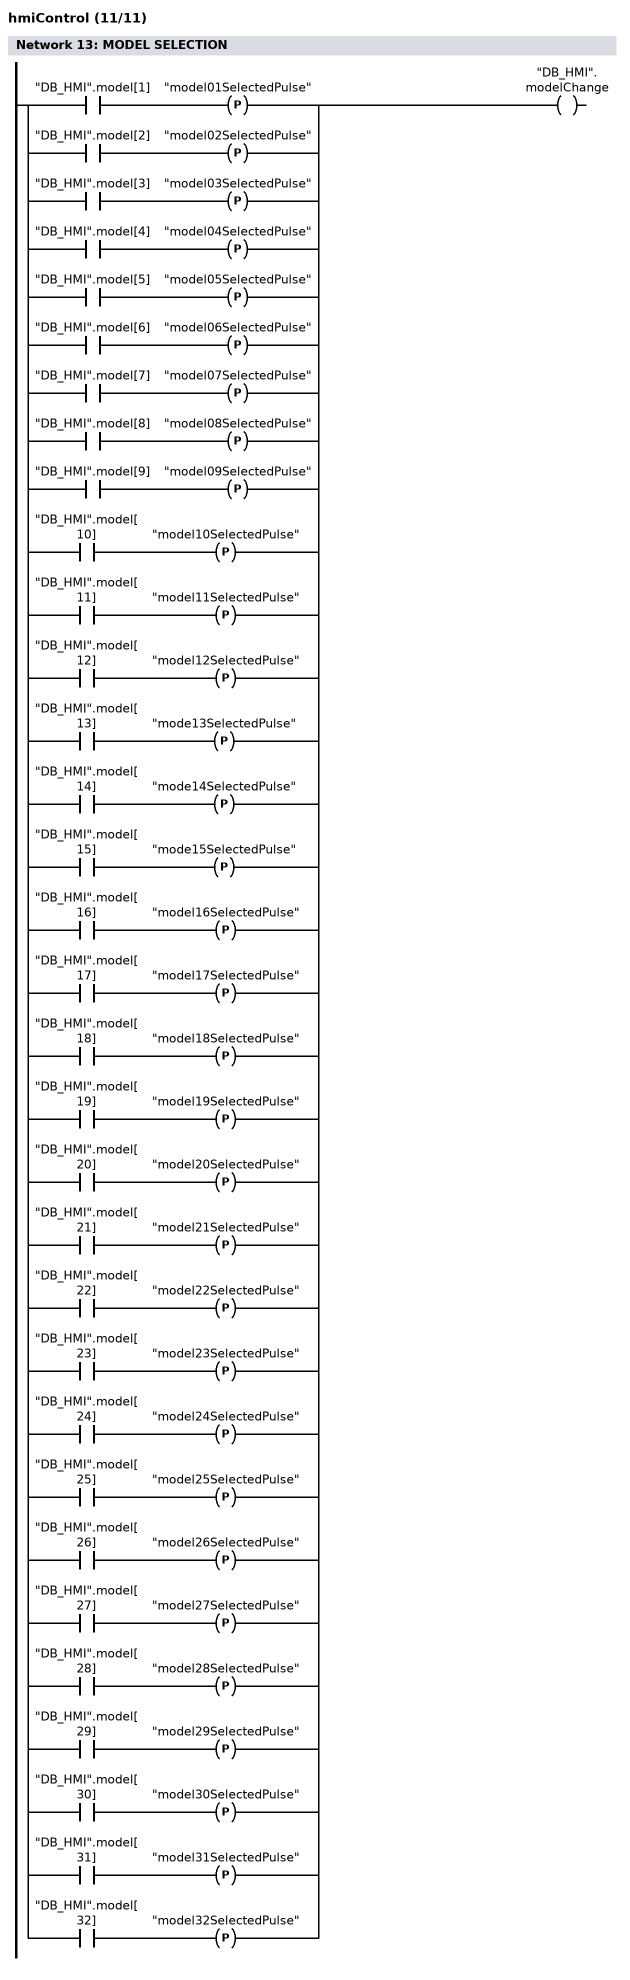
   RUNG wire#powerrail
      Contact( "DB_HMI".model[1] )
      P_Trig( "model01SelectedPulse" )
      wire#w1
      Coil( "DB_HMI".modelChange )
   END_RUNG
   RUNG wire#powerrail
      Contact( "DB_HMI".model[2] )
      P_Trig( "model02SelectedPulse" )
   END_RUNG wire#w1
   RUNG wire#powerrail
      Contact( "DB_HMI".model[3] )
      P_Trig( "model03SelectedPulse" )
   END_RUNG wire#w1
   RUNG wire#powerrail
      Contact( "DB_HMI".model[4] )
      P_Trig( "model04SelectedPulse" )
   END_RUNG wire#w1
   RUNG wire#powerrail
      Contact( "DB_HMI".model[5] )
      P_Trig( "model05SelectedPulse" )
   END_RUNG wire#w1
   RUNG wire#powerrail
      Contact( "DB_HMI".model[6] )
      P_Trig( "model06SelectedPulse" )
   END_RUNG wire#w1
   RUNG wire#powerrail
      Contact( "DB_HMI".model[7] )
      P_Trig( "model07SelectedPulse" )
   END_RUNG wire#w1
   RUNG wire#powerrail
      Contact( "DB_HMI".model[8] )
      P_Trig( "model08SelectedPulse" )
   END_RUNG wire#w1
   RUNG wire#powerrail
      Contact( "DB_HMI".model[9] )
      P_Trig( "model09SelectedPulse" )
   END_RUNG wire#w1
   RUNG wire#powerrail
      Contact( "DB_HMI".model[10] )
      P_Trig( "model10SelectedPulse" )
   END_RUNG wire#w1
   RUNG wire#powerrail
      Contact( "DB_HMI".model[11] )
      P_Trig( "model11SelectedPulse" )
   END_RUNG wire#w1
   RUNG wire#powerrail
      Contact( "DB_HMI".model[12] )
      P_Trig( "model12SelectedPulse" )
   END_RUNG wire#w1
   RUNG wire#powerrail
      Contact( "DB_HMI".model[13] )
      P_Trig( "mode13SelectedPulse" )
   END_RUNG wire#w1
   RUNG wire#powerrail
      Contact( "DB_HMI".model[14] )
      P_Trig( "mode14SelectedPulse" )
   END_RUNG wire#w1
   RUNG wire#powerrail
      Contact( "DB_HMI".model[15] )
      P_Trig( "mode15SelectedPulse" )
   END_RUNG wire#w1
   RUNG wire#powerrail
      Contact( "DB_HMI".model[16] )
      P_Trig( "model16SelectedPulse" )
   END_RUNG wire#w1
   RUNG wire#powerrail
      Contact( "DB_HMI".model[17] )
      P_Trig( "model17SelectedPulse" )
   END_RUNG wire#w1
   RUNG wire#powerrail
      Contact( "DB_HMI".model[18] )
      P_Trig( "model18SelectedPulse" )
   END_RUNG wire#w1
   RUNG wire#powerrail
      Contact( "DB_HMI".model[19] )
      P_Trig( "model19SelectedPulse" )
   END_RUNG wire#w1
   RUNG wire#powerrail
      Contact( "DB_HMI".model[20] )
      P_Trig( "model20SelectedPulse" )
   END_RUNG wire#w1
   RUNG wire#powerrail
      Contact( "DB_HMI".model[21] )
      P_Trig( "model21SelectedPulse" )
   END_RUNG wire#w1
   RUNG wire#powerrail
      Contact( "DB_HMI".model[22] )
      P_Trig( "model22SelectedPulse" )
   END_RUNG wire#w1
   RUNG wire#powerrail
      Contact( "DB_HMI".model[23] )
      P_Trig( "model23SelectedPulse" )
   END_RUNG wire#w1
   RUNG wire#powerrail
      Contact( "DB_HMI".model[24] )
      P_Trig( "model24SelectedPulse" )
   END_RUNG wire#w1
   RUNG wire#powerrail
      Contact( "DB_HMI".model[25] )
      P_Trig( "model25SelectedPulse" )
   END_RUNG wire#w1
   RUNG wire#powerrail
      Contact( "DB_HMI".model[26] )
      P_Trig( "model26SelectedPulse" )
   END_RUNG wire#w1
   RUNG wire#powerrail
      Contact( "DB_HMI".model[27] )
      P_Trig( "model27SelectedPulse" )
   END_RUNG wire#w1
   RUNG wire#powerrail
      Contact( "DB_HMI".model[28] )
      P_Trig( "model28SelectedPulse" )
   END_RUNG wire#w1
   RUNG wire#powerrail
      Contact( "DB_HMI".model[29] )
      P_Trig( "model29SelectedPulse" )
   END_RUNG wire#w1
   RUNG wire#powerrail
      Contact( "DB_HMI".model[30] )
      P_Trig( "model30SelectedPulse" )
   END_RUNG wire#w1
   RUNG wire#powerrail
      Contact( "DB_HMI".model[31] )
      P_Trig( "model31SelectedPulse" )
   END_RUNG wire#w1
   RUNG wire#powerrail
      Contact( "DB_HMI".model[32] )
      P_Trig( "model32SelectedPulse" )
   END_RUNG wire#w1
   // the same network as SCL:
   #_w1 := "DB_HMI".model[1] AND NOT "model01SelectedPulse";   // rising edge
   "model01SelectedPulse" := "DB_HMI".model[1];
   #_w2 := "DB_HMI".model[2] AND NOT "model02SelectedPulse";   // rising edge
   "model02SelectedPulse" := "DB_HMI".model[2];
   #_w3 := "DB_HMI".model[3] AND NOT "model03SelectedPulse";   // rising edge
   "model03SelectedPulse" := "DB_HMI".model[3];
   #_w4 := "DB_HMI".model[4] AND NOT "model04SelectedPulse";   // rising edge
   "model04SelectedPulse" := "DB_HMI".model[4];
   #_w5 := "DB_HMI".model[5] AND NOT "model05SelectedPulse";   // rising edge
   "model05SelectedPulse" := "DB_HMI".model[5];
   #_w6 := "DB_HMI".model[6] AND NOT "model06SelectedPulse";   // rising edge
   "model06SelectedPulse" := "DB_HMI".model[6];
   #_w7 := "DB_HMI".model[7] AND NOT "model07SelectedPulse";   // rising edge
   "model07SelectedPulse" := "DB_HMI".model[7];
   #_w8 := "DB_HMI".model[8] AND NOT "model08SelectedPulse";   // rising edge
   "model08SelectedPulse" := "DB_HMI".model[8];
   #_w9 := "DB_HMI".model[9] AND NOT "model09SelectedPulse";   // rising edge
   "model09SelectedPulse" := "DB_HMI".model[9];
   #_w10 := "DB_HMI".model[10] AND NOT "model10SelectedPulse";   // rising edge
   "model10SelectedPulse" := "DB_HMI".model[10];
   #_w11 := "DB_HMI".model[11] AND NOT "model11SelectedPulse";   // rising edge
   "model11SelectedPulse" := "DB_HMI".model[11];
   #_w12 := "DB_HMI".model[12] AND NOT "model12SelectedPulse";   // rising edge
   "model12SelectedPulse" := "DB_HMI".model[12];
   #_w13 := "DB_HMI".model[13] AND NOT "mode13SelectedPulse";   // rising edge
   "mode13SelectedPulse" := "DB_HMI".model[13];
   #_w14 := "DB_HMI".model[14] AND NOT "mode14SelectedPulse";   // rising edge
   "mode14SelectedPulse" := "DB_HMI".model[14];
   #_w15 := "DB_HMI".model[15] AND NOT "mode15SelectedPulse";   // rising edge
   "mode15SelectedPulse" := "DB_HMI".model[15];
   #_w16 := "DB_HMI".model[16] AND NOT "model16SelectedPulse";   // rising edge
   "model16SelectedPulse" := "DB_HMI".model[16];
   #_w17 := "DB_HMI".model[17] AND NOT "model17SelectedPulse";   // rising edge
   "model17SelectedPulse" := "DB_HMI".model[17];
   #_w18 := "DB_HMI".model[18] AND NOT "model18SelectedPulse";   // rising edge
   "model18SelectedPulse" := "DB_HMI".model[18];
   #_w19 := "DB_HMI".model[19] AND NOT "model19SelectedPulse";   // rising edge
   "model19SelectedPulse" := "DB_HMI".model[19];
   #_w20 := "DB_HMI".model[20] AND NOT "model20SelectedPulse";   // rising edge
   "model20SelectedPulse" := "DB_HMI".model[20];
   #_w21 := "DB_HMI".model[21] AND NOT "model21SelectedPulse";   // rising edge
   "model21SelectedPulse" := "DB_HMI".model[21];
   #_w22 := "DB_HMI".model[22] AND NOT "model22SelectedPulse";   // rising edge
   "model22SelectedPulse" := "DB_HMI".model[22];
   #_w23 := "DB_HMI".model[23] AND NOT "model23SelectedPulse";   // rising edge
   "model23SelectedPulse" := "DB_HMI".model[23];
   #_w24 := "DB_HMI".model[24] AND NOT "model24SelectedPulse";   // rising edge
   "model24SelectedPulse" := "DB_HMI".model[24];
   #_w25 := "DB_HMI".model[25] AND NOT "model25SelectedPulse";   // rising edge
   "model25SelectedPulse" := "DB_HMI".model[25];
   #_w26 := "DB_HMI".model[26] AND NOT "model26SelectedPulse";   // rising edge
   "model26SelectedPulse" := "DB_HMI".model[26];
   #_w27 := "DB_HMI".model[27] AND NOT "model27SelectedPulse";   // rising edge
   "model27SelectedPulse" := "DB_HMI".model[27];
   #_w28 := "DB_HMI".model[28] AND NOT "model28SelectedPulse";   // rising edge
   "model28SelectedPulse" := "DB_HMI".model[28];
   #_w29 := "DB_HMI".model[29] AND NOT "model29SelectedPulse";   // rising edge
   "model29SelectedPulse" := "DB_HMI".model[29];
   #_w30 := "DB_HMI".model[30] AND NOT "model30SelectedPulse";   // rising edge
   "model30SelectedPulse" := "DB_HMI".model[30];
   #_w31 := "DB_HMI".model[31] AND NOT "model31SelectedPulse";   // rising edge
   "model31SelectedPulse" := "DB_HMI".model[31];
   #_w32 := "DB_HMI".model[32] AND NOT "model32SelectedPulse";   // rising edge
   "model32SelectedPulse" := "DB_HMI".model[32];
   "DB_HMI".modelChange := #_w1 OR #_w2 OR #_w3 OR #_w4 OR #_w5 OR #_w6 OR #_w7 OR #_w8 OR #_w9 OR #_w10 OR #_w11 OR #_w12 OR #_w13 OR #_w14 OR #_w15 OR #_w16 OR #_w17 OR #_w18 OR #_w19 OR #_w20 OR #_w21 OR #_w22 OR #_w23 OR #_w24 OR #_w25 OR #_w26 OR #_w27 OR #_w28 OR #_w29 OR #_w30 OR #_w31 OR #_w32;
END_REGION
END_FUNCTION

FUNCTION "MODE" : Void   // FC4, LAD
{ S7_Optimized_Access := 'TRUE' }
VERSION : 0.1
// stored: AutoNumber true, IsIECCheckEnabled false, SetENOAutomatically false, UDAEnableTagReadback false
   VAR_TEMP
      f7 : Bool;
      BF7 : Bool;
   END_VAR
BEGIN

REGION Network 1: MODE CHANGE
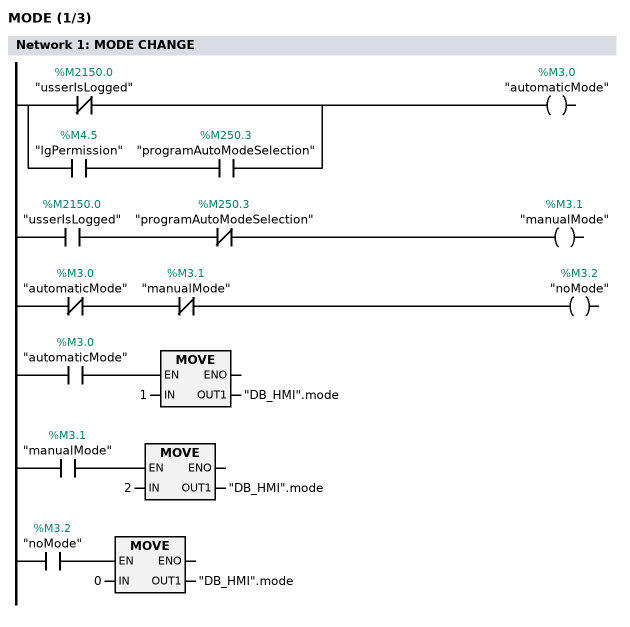
   RUNG wire#powerrail
      I_Contact( "usserIsLogged" )
      wire#w1
      Coil( "automaticMode" )
   END_RUNG
   RUNG wire#powerrail
      Contact( "lgPermission" )
      Contact( "programAutoModeSelection" )
   END_RUNG wire#w1
   RUNG wire#powerrail
      Contact( "usserIsLogged" )
      I_Contact( "programAutoModeSelection" )
      Coil( "manualMode" )
   END_RUNG
   RUNG wire#powerrail
      I_Contact( "automaticMode" )
      I_Contact( "manualMode" )
      Coil( "noMode" )
   END_RUNG
   RUNG wire#powerrail
      Contact( "automaticMode" )
      Move(in := 1, out1 => "DB_HMI".mode)
   END_RUNG
   RUNG wire#powerrail
      Contact( "manualMode" )
      Move(in := 2, out1 => "DB_HMI".mode)
   END_RUNG
   RUNG wire#powerrail
      Contact( "noMode" )
      Move(in := 0, out1 => "DB_HMI".mode)
   END_RUNG
   // the same network as SCL:
   "automaticMode" := NOT "usserIsLogged" OR ("lgPermission" AND "programAutoModeSelection");
   "manualMode" := "usserIsLogged" AND NOT "programAutoModeSelection";
   "noMode" := NOT "automaticMode" AND NOT "manualMode";
   IF "automaticMode" THEN "DB_HMI".mode := 1; END_IF;
   IF "manualMode" THEN "DB_HMI".mode := 2; END_IF;
   IF "noMode" THEN "DB_HMI".mode := 0; END_IF;
END_REGION

REGION Network 2: MODEL SELECTION
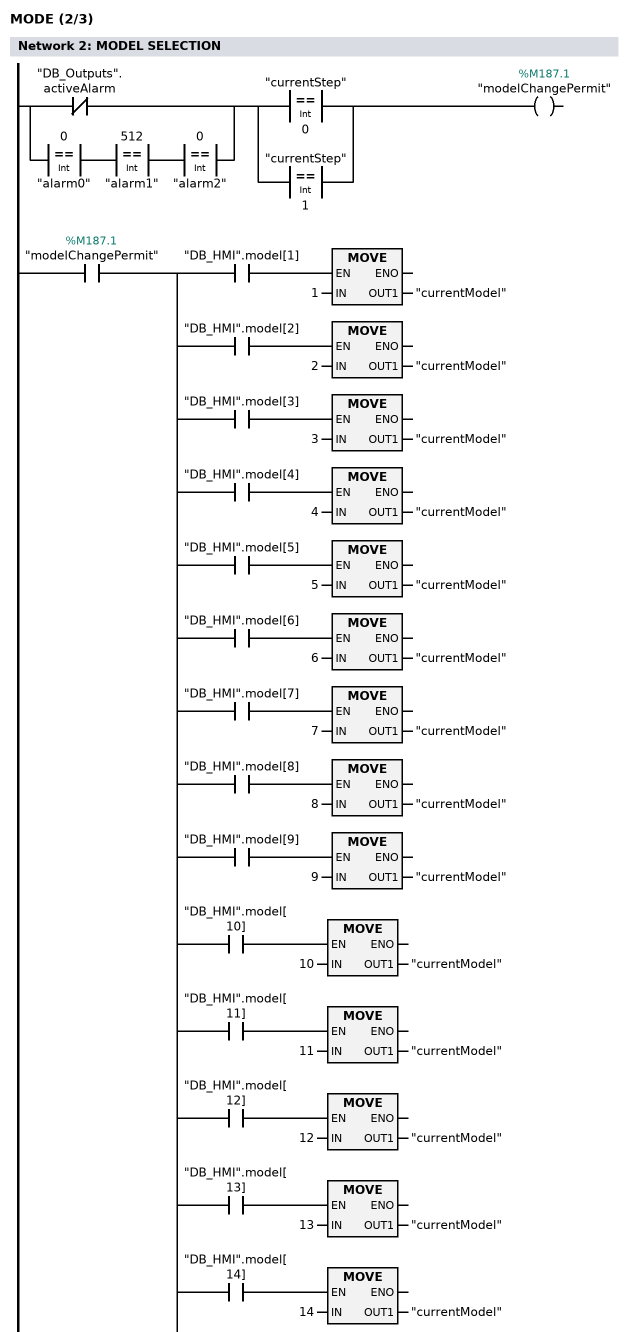
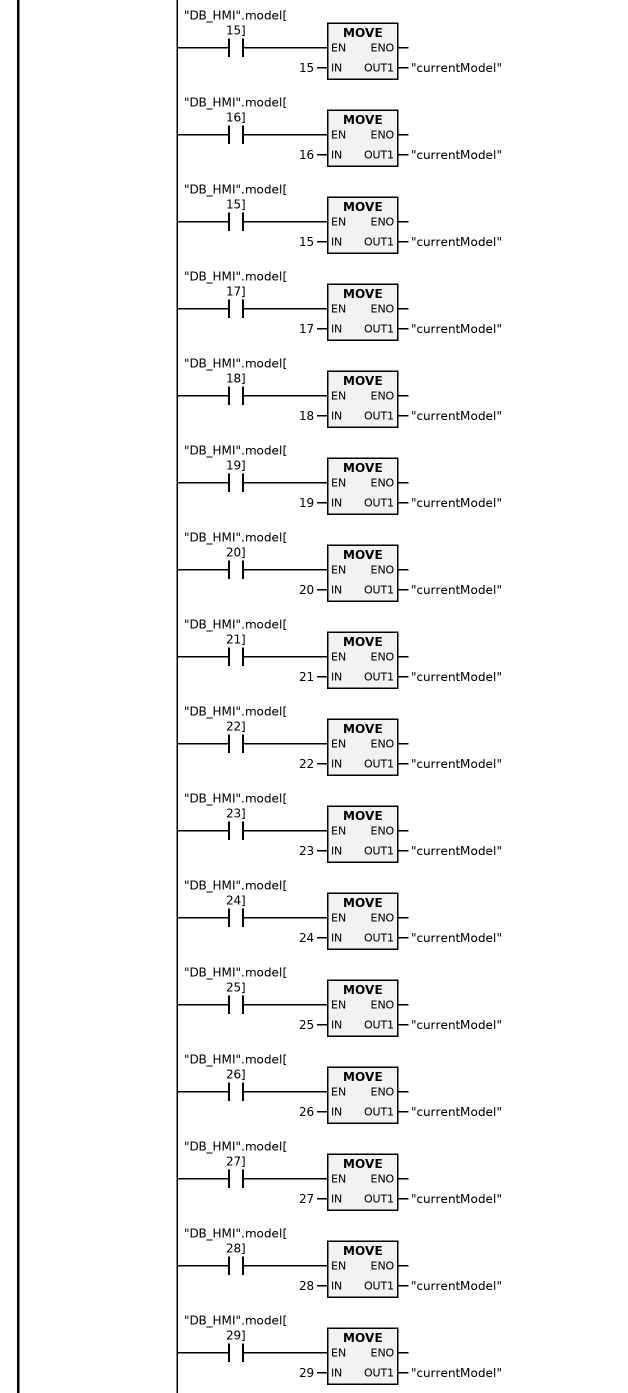
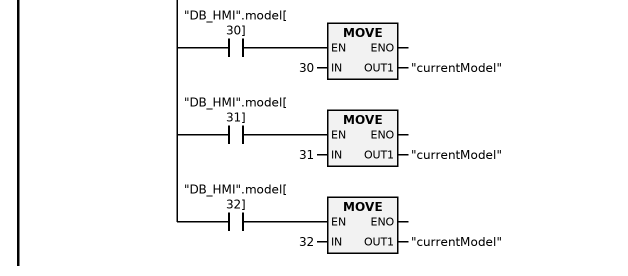
   RUNG wire#powerrail
      I_Contact( "DB_Outputs".activeAlarm )
      wire#w1
      { S7_Templates := "SrcType := Int" } EQ_Contact(in1 := "currentStep", in2 := 0)
      wire#w2
      Coil( "modelChangePermit" )
   END_RUNG
   RUNG wire#powerrail
      { S7_Templates := "SrcType := Int" } EQ_Contact(in1 := 0, in2 := "alarm0")
      { S7_Templates := "SrcType := Int" } EQ_Contact(in1 := 512, in2 := "alarm1")
      { S7_Templates := "SrcType := Int" } EQ_Contact(in1 := 0, in2 := "alarm2")
   END_RUNG wire#w1
   RUNG wire#w1
      { S7_Templates := "SrcType := Int" } EQ_Contact(in1 := "currentStep", in2 := 1)
   END_RUNG wire#w2
   RUNG wire#powerrail
      Contact( "modelChangePermit" )
      wire#w3
      Contact( "DB_HMI".model[1] )
      Move(in := 1, out1 => "currentModel")
   END_RUNG
   RUNG wire#w3
      Contact( "DB_HMI".model[2] )
      Move(in := 2, out1 => "currentModel")
   END_RUNG
   RUNG wire#w3
      Contact( "DB_HMI".model[3] )
      Move(in := 3, out1 => "currentModel")
   END_RUNG
   RUNG wire#w3
      Contact( "DB_HMI".model[4] )
      Move(in := 4, out1 => "currentModel")
   END_RUNG
   RUNG wire#w3
      Contact( "DB_HMI".model[5] )
      Move(in := 5, out1 => "currentModel")
   END_RUNG
   RUNG wire#w3
      Contact( "DB_HMI".model[6] )
      Move(in := 6, out1 => "currentModel")
   END_RUNG
   RUNG wire#w3
      Contact( "DB_HMI".model[7] )
      Move(in := 7, out1 => "currentModel")
   END_RUNG
   RUNG wire#w3
      Contact( "DB_HMI".model[8] )
      Move(in := 8, out1 => "currentModel")
   END_RUNG
   RUNG wire#w3
      Contact( "DB_HMI".model[9] )
      Move(in := 9, out1 => "currentModel")
   END_RUNG
   RUNG wire#w3
      Contact( "DB_HMI".model[10] )
      Move(in := 10, out1 => "currentModel")
   END_RUNG
   RUNG wire#w3
      Contact( "DB_HMI".model[11] )
      Move(in := 11, out1 => "currentModel")
   END_RUNG
   RUNG wire#w3
      Contact( "DB_HMI".model[12] )
      Move(in := 12, out1 => "currentModel")
   END_RUNG
   RUNG wire#w3
      Contact( "DB_HMI".model[13] )
      Move(in := 13, out1 => "currentModel")
   END_RUNG
   RUNG wire#w3
      Contact( "DB_HMI".model[14] )
      Move(in := 14, out1 => "currentModel")
   END_RUNG
   RUNG wire#w3
      Contact( "DB_HMI".model[15] )
      Move(in := 15, out1 => "currentModel")
   END_RUNG
   RUNG wire#w3
      Contact( "DB_HMI".model[16] )
      Move(in := 16, out1 => "currentModel")
   END_RUNG
   RUNG wire#w3
      Contact( "DB_HMI".model[15] )
      Move(in := 15, out1 => "currentModel")
   END_RUNG
   RUNG wire#w3
      Contact( "DB_HMI".model[17] )
      Move(in := 17, out1 => "currentModel")
   END_RUNG
   RUNG wire#w3
      Contact( "DB_HMI".model[18] )
      Move(in := 18, out1 => "currentModel")
   END_RUNG
   RUNG wire#w3
      Contact( "DB_HMI".model[19] )
      Move(in := 19, out1 => "currentModel")
   END_RUNG
   RUNG wire#w3
      Contact( "DB_HMI".model[20] )
      Move(in := 20, out1 => "currentModel")
   END_RUNG
   RUNG wire#w3
      Contact( "DB_HMI".model[21] )
      Move(in := 21, out1 => "currentModel")
   END_RUNG
   RUNG wire#w3
      Contact( "DB_HMI".model[22] )
      Move(in := 22, out1 => "currentModel")
   END_RUNG
   RUNG wire#w3
      Contact( "DB_HMI".model[23] )
      Move(in := 23, out1 => "currentModel")
   END_RUNG
   RUNG wire#w3
      Contact( "DB_HMI".model[24] )
      Move(in := 24, out1 => "currentModel")
   END_RUNG
   RUNG wire#w3
      Contact( "DB_HMI".model[25] )
      Move(in := 25, out1 => "currentModel")
   END_RUNG
   RUNG wire#w3
      Contact( "DB_HMI".model[26] )
      Move(in := 26, out1 => "currentModel")
   END_RUNG
   RUNG wire#w3
      Contact( "DB_HMI".model[27] )
      Move(in := 27, out1 => "currentModel")
   END_RUNG
   RUNG wire#w3
      Contact( "DB_HMI".model[28] )
      Move(in := 28, out1 => "currentModel")
   END_RUNG
   RUNG wire#w3
      Contact( "DB_HMI".model[29] )
      Move(in := 29, out1 => "currentModel")
   END_RUNG
   RUNG wire#w3
      Contact( "DB_HMI".model[30] )
      Move(in := 30, out1 => "currentModel")
   END_RUNG
   RUNG wire#w3
      Contact( "DB_HMI".model[31] )
      Move(in := 31, out1 => "currentModel")
   END_RUNG
   RUNG wire#w3
      Contact( "DB_HMI".model[32] )
      Move(in := 32, out1 => "currentModel")
   END_RUNG
   // the same network as SCL:
   "modelChangePermit" := (NOT "DB_Outputs".activeAlarm OR ((0 = "alarm0") AND (512 = "alarm1") AND (0 = "alarm2"))) AND (("currentStep" = 0) OR ("currentStep" = 1));
   IF "modelChangePermit" AND "DB_HMI".model[1] THEN "currentModel" := 1; END_IF;
   IF "modelChangePermit" AND "DB_HMI".model[2] THEN "currentModel" := 2; END_IF;
   IF "modelChangePermit" AND "DB_HMI".model[3] THEN "currentModel" := 3; END_IF;
   IF "modelChangePermit" AND "DB_HMI".model[4] THEN "currentModel" := 4; END_IF;
   IF "modelChangePermit" AND "DB_HMI".model[5] THEN "currentModel" := 5; END_IF;
   IF "modelChangePermit" AND "DB_HMI".model[6] THEN "currentModel" := 6; END_IF;
   IF "modelChangePermit" AND "DB_HMI".model[7] THEN "currentModel" := 7; END_IF;
   IF "modelChangePermit" AND "DB_HMI".model[8] THEN "currentModel" := 8; END_IF;
   IF "modelChangePermit" AND "DB_HMI".model[9] THEN "currentModel" := 9; END_IF;
   IF "modelChangePermit" AND "DB_HMI".model[10] THEN "currentModel" := 10; END_IF;
   IF "modelChangePermit" AND "DB_HMI".model[11] THEN "currentModel" := 11; END_IF;
   IF "modelChangePermit" AND "DB_HMI".model[12] THEN "currentModel" := 12; END_IF;
   IF "modelChangePermit" AND "DB_HMI".model[13] THEN "currentModel" := 13; END_IF;
   IF "modelChangePermit" AND "DB_HMI".model[14] THEN "currentModel" := 14; END_IF;
   IF "modelChangePermit" AND "DB_HMI".model[15] THEN "currentModel" := 15; END_IF;
   IF "modelChangePermit" AND "DB_HMI".model[16] THEN "currentModel" := 16; END_IF;
   IF "modelChangePermit" AND "DB_HMI".model[15] THEN "currentModel" := 15; END_IF;
   IF "modelChangePermit" AND "DB_HMI".model[17] THEN "currentModel" := 17; END_IF;
   IF "modelChangePermit" AND "DB_HMI".model[18] THEN "currentModel" := 18; END_IF;
   IF "modelChangePermit" AND "DB_HMI".model[19] THEN "currentModel" := 19; END_IF;
   IF "modelChangePermit" AND "DB_HMI".model[20] THEN "currentModel" := 20; END_IF;
   IF "modelChangePermit" AND "DB_HMI".model[21] THEN "currentModel" := 21; END_IF;
   IF "modelChangePermit" AND "DB_HMI".model[22] THEN "currentModel" := 22; END_IF;
   IF "modelChangePermit" AND "DB_HMI".model[23] THEN "currentModel" := 23; END_IF;
   IF "modelChangePermit" AND "DB_HMI".model[24] THEN "currentModel" := 24; END_IF;
   IF "modelChangePermit" AND "DB_HMI".model[25] THEN "currentModel" := 25; END_IF;
   IF "modelChangePermit" AND "DB_HMI".model[26] THEN "currentModel" := 26; END_IF;
   IF "modelChangePermit" AND "DB_HMI".model[27] THEN "currentModel" := 27; END_IF;
   IF "modelChangePermit" AND "DB_HMI".model[28] THEN "currentModel" := 28; END_IF;
   IF "modelChangePermit" AND "DB_HMI".model[29] THEN "currentModel" := 29; END_IF;
   IF "modelChangePermit" AND "DB_HMI".model[30] THEN "currentModel" := 30; END_IF;
   IF "modelChangePermit" AND "DB_HMI".model[31] THEN "currentModel" := 31; END_IF;
   IF "modelChangePermit" AND "DB_HMI".model[32] THEN "currentModel" := 32; END_IF;
END_REGION

REGION Network 3: GAP LEADER HMI MODE
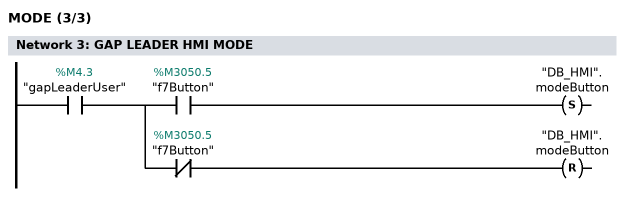
   RUNG wire#powerrail
      Contact( "gapLeaderUser" )
      wire#w1
      Contact( "f7Button" )
      S_Coil( "DB_HMI".modeButton )
   END_RUNG
   RUNG wire#w1
      I_Contact( "f7Button" )
      R_Coil( "DB_HMI".modeButton )
   END_RUNG
   // the same network as SCL:
   IF "gapLeaderUser" AND "f7Button" THEN "DB_HMI".modeButton := TRUE; END_IF;
   IF "gapLeaderUser" AND NOT "f7Button" THEN "DB_HMI".modeButton := FALSE; END_IF;
END_REGION
END_FUNCTION

FUNCTION "MISC" : Void   // FC5, LAD
{ S7_Optimized_Access := 'TRUE' }
VERSION : 0.1
// stored: AutoNumber true, IsIECCheckEnabled false, SetENOAutomatically false, UDAEnableTagReadback false
   VAR_TEMP
      INTERMITENTE : Bool;
      RESETEADO : Bool;
      RESULT_2 : UInt;
      Result_3 : Int;
   END_VAR
   VAR_TEMP   // added for the SCL form of the ladder/FBD networks
      _w1 : Bool;
      _w2 : Bool;
      _w3 : Bool;
      _w4 : Bool;
   END_VAR
BEGIN

REGION Network 1: HMI OPTIONS BUTTON SHUTOFF
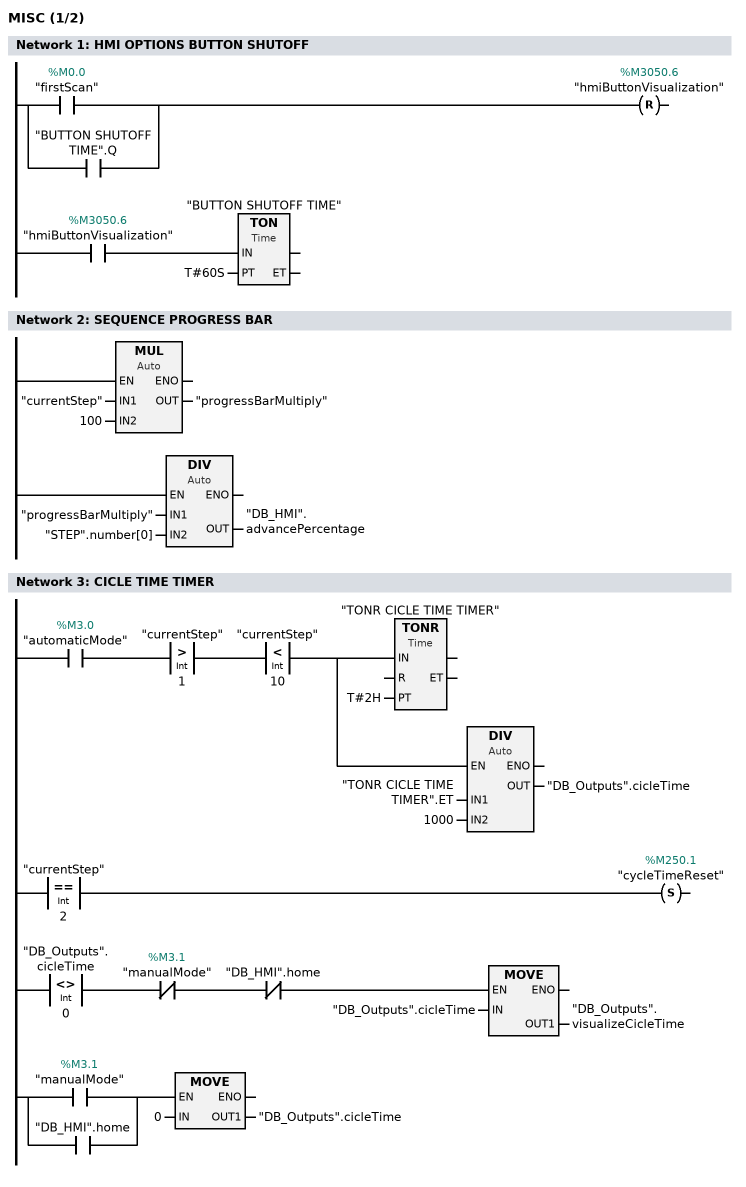
   RUNG wire#powerrail
      Contact( "firstScan" )
      wire#w1
      R_Coil( "hmiButtonVisualization" )
   END_RUNG
   RUNG wire#powerrail
      Contact( "BUTTON SHUTOFF TIME".Q )
   END_RUNG wire#w1
   RUNG wire#powerrail
      Contact( "hmiButtonVisualization" )
      { S7_Templates := "time_type := Time" } "BUTTON SHUTOFF TIME".TON(pt := T#60S, et =>)
   END_RUNG
   // the same network as SCL:
   IF "firstScan" OR "BUTTON SHUTOFF TIME".Q THEN "hmiButtonVisualization" := FALSE; END_IF;
   "BUTTON SHUTOFF TIME".TON(IN := "hmiButtonVisualization", PT := T#60S);
END_REGION

REGION Network 2: SEQUENCE PROGRESS BAR
   RUNG wire#powerrail
      Mul(in1 := "currentStep", in2 := 100, out => "progressBarMultiply")
   END_RUNG
   RUNG wire#powerrail
      Div(in1 := "progressBarMultiply", in2 := "STEP".number[0], out => "DB_HMI".advancePercentage)
   END_RUNG
   // the same network as SCL:
   "progressBarMultiply" := "currentStep" * 100;
   "DB_HMI".advancePercentage := "progressBarMultiply" / "STEP".number[0];
END_REGION

REGION Network 3: CICLE TIME TIMER
   RUNG wire#powerrail
      Contact( "automaticMode" )
      { S7_Templates := "SrcType := Int" } GT_Contact(in1 := "currentStep", in2 := 1)
      { S7_Templates := "SrcType := Int" } LT_Contact(in1 := "currentStep", in2 := 10)
      wire#w1
      { S7_Templates := "time_type := Time" } "TONR CICLE TIME TIMER".TONR(r :=, pt := T#2H, et =>)
   END_RUNG
   RUNG wire#w1
      Div(in1 := "TONR CICLE TIME TIMER".ET, in2 := 1000, out => "DB_Outputs".cicleTime)
   END_RUNG
   RUNG wire#powerrail
      { S7_Templates := "SrcType := Int" } EQ_Contact(in1 := "currentStep", in2 := 2)
      S_Coil( "cycleTimeReset" )
   END_RUNG
   RUNG wire#powerrail
      { S7_Templates := "SrcType := Int" } NE_Contact(in1 := "DB_Outputs".cicleTime, in2 := 0)
      I_Contact( "manualMode" )
      I_Contact( "DB_HMI".home )
      Move(in := "DB_Outputs".cicleTime, out1 => "DB_Outputs".visualizeCicleTime)
   END_RUNG
   RUNG wire#powerrail
      Contact( "manualMode" )
      wire#w2
      Move(in := 0, out1 => "DB_Outputs".cicleTime)
   END_RUNG
   RUNG wire#powerrail
      Contact( "DB_HMI".home )
   END_RUNG wire#w2
   // the same network as SCL:
   #_w1 := "automaticMode" AND ("currentStep" > 1) AND ("currentStep" < 10);
   "TONR CICLE TIME TIMER".TONR(IN := #_w1, PT := T#2H);
   IF #_w1 THEN "DB_Outputs".cicleTime := "TONR CICLE TIME TIMER".ET / 1000; END_IF;
   IF "currentStep" = 2 THEN "cycleTimeReset" := TRUE; END_IF;
   IF ("DB_Outputs".cicleTime <> 0) AND NOT "manualMode" AND NOT "DB_HMI".home THEN
       "DB_Outputs".visualizeCicleTime := "DB_Outputs".cicleTime;
   END_IF;
   IF "manualMode" OR "DB_HMI".home THEN "DB_Outputs".cicleTime := 0; END_IF;
END_REGION

REGION Network 4: STEP CHANGE TIMER
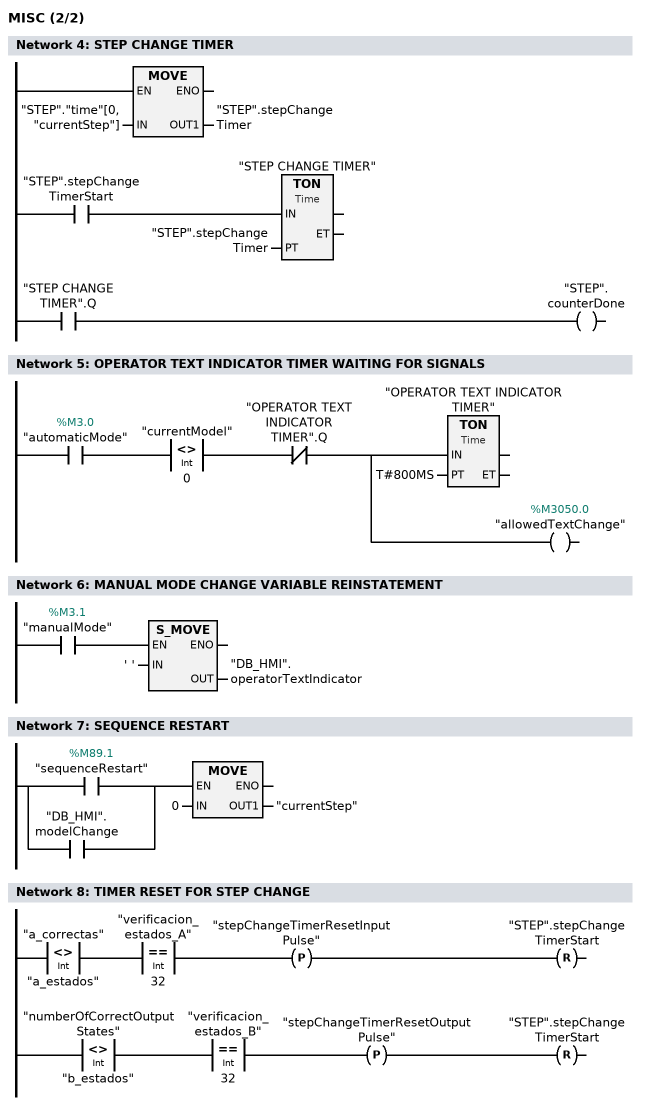
   RUNG wire#powerrail
      Move(in := "STEP"."time"[0, "currentStep"], out1 => "STEP".stepChangeTimer)
   END_RUNG
   RUNG wire#powerrail
      Contact( "STEP".stepChangeTimerStart )
      { S7_Templates := "time_type := Time" } "STEP CHANGE TIMER".TON(pt := "STEP".stepChangeTimer, et =>)
   END_RUNG
   RUNG wire#powerrail
      Contact( "STEP CHANGE TIMER".Q )
      Coil( "STEP".counterDone )
   END_RUNG
   // the same network as SCL:
   "STEP".stepChangeTimer := "STEP"."time"[0, "currentStep"];
   "STEP CHANGE TIMER".TON(IN := "STEP".stepChangeTimerStart, PT := "STEP".stepChangeTimer);
   "STEP".counterDone := "STEP CHANGE TIMER".Q;
END_REGION

REGION Network 5: OPERATOR TEXT INDICATOR TIMER WAITING FOR SIGNALS
   RUNG wire#powerrail
      Contact( "automaticMode" )
      { S7_Templates := "SrcType := Int" } NE_Contact(in1 := "currentModel", in2 := 0)
      I_Contact( "OPERATOR TEXT INDICATOR TIMER".Q )
      wire#w1
      { S7_Templates := "time_type := Time" } "OPERATOR TEXT INDICATOR TIMER".TON(pt := T#800MS, et =>)
   END_RUNG
   RUNG wire#w1
      Coil( "allowedTextChange" )
   END_RUNG
   // the same network as SCL:
   #_w1 := "automaticMode" AND ("currentModel" <> 0) AND NOT "OPERATOR TEXT INDICATOR TIMER".Q;
   "OPERATOR TEXT INDICATOR TIMER".TON(IN := #_w1, PT := T#800MS);
   "allowedTextChange" := #_w1;
END_REGION

REGION Network 6: MANUAL MODE CHANGE VARIABLE REINSTATEMENT
   RUNG wire#powerrail
      Contact( "manualMode" )
      S_Move(in := ' ', out => "DB_HMI".operatorTextIndicator)
   END_RUNG
   // the same network as SCL:
   IF "manualMode" THEN "DB_HMI".operatorTextIndicator := ' '; END_IF;
END_REGION

REGION Network 7: SEQUENCE RESTART
   RUNG wire#powerrail
      Contact( "sequenceRestart" )
      wire#w1
      Move(in := 0, out1 => "currentStep")
   END_RUNG
   RUNG wire#powerrail
      Contact( "DB_HMI".modelChange )
   END_RUNG wire#w1
   // the same network as SCL:
   IF "sequenceRestart" OR "DB_HMI".modelChange THEN "currentStep" := 0; END_IF;
END_REGION

REGION Network 8: TIMER RESET FOR STEP CHANGE
   RUNG wire#powerrail
      { S7_Templates := "SrcType := Int" } NE_Contact(in1 := "a_correctas", in2 := "a_estados")
      { S7_Templates := "SrcType := Int" } EQ_Contact(in1 := "verificacion_estados_A", in2 := 32)
      P_Trig( "stepChangeTimerResetInputPulse" )
      R_Coil( "STEP".stepChangeTimerStart )
   END_RUNG
   RUNG wire#powerrail
      { S7_Templates := "SrcType := Int" } NE_Contact(in1 := "numberOfCorrectOutputStates", in2 := "b_estados")
      { S7_Templates := "SrcType := Int" } EQ_Contact(in1 := "verificacion_estados_B", in2 := 32)
      P_Trig( "stepChangeTimerResetOutputPulse" )
      R_Coil( "STEP".stepChangeTimerStart )
   END_RUNG
   // the same network as SCL:
   #_w1 := ("a_correctas" <> "a_estados") AND ("verificacion_estados_A" = 32);
   #_w2 := #_w1 AND NOT "stepChangeTimerResetInputPulse";   // rising edge
   "stepChangeTimerResetInputPulse" := #_w1;
   IF #_w2 THEN "STEP".stepChangeTimerStart := FALSE; END_IF;
   #_w3 := ("numberOfCorrectOutputStates" <> "b_estados") AND ("verificacion_estados_B" = 32);
   #_w4 := #_w3 AND NOT "stepChangeTimerResetOutputPulse";   // rising edge
   "stepChangeTimerResetOutputPulse" := #_w3;
   IF #_w4 THEN "STEP".stepChangeTimerStart := FALSE; END_IF;
END_REGION
END_FUNCTION

FUNCTION "MODIFY RECIPE" : Void   // FC6, LAD
{ S7_Optimized_Access := 'TRUE' }
VERSION : 0.1
// stored: AutoNumber true, IsIECCheckEnabled false, SetENOAutomatically false, UDAEnableTagReadback false
   VAR_TEMP   // added for the SCL form of the ladder/FBD networks
      _w1 : Bool;
      _w2 : Bool;
   END_VAR
BEGIN

REGION Network 1: ERASE A STEP
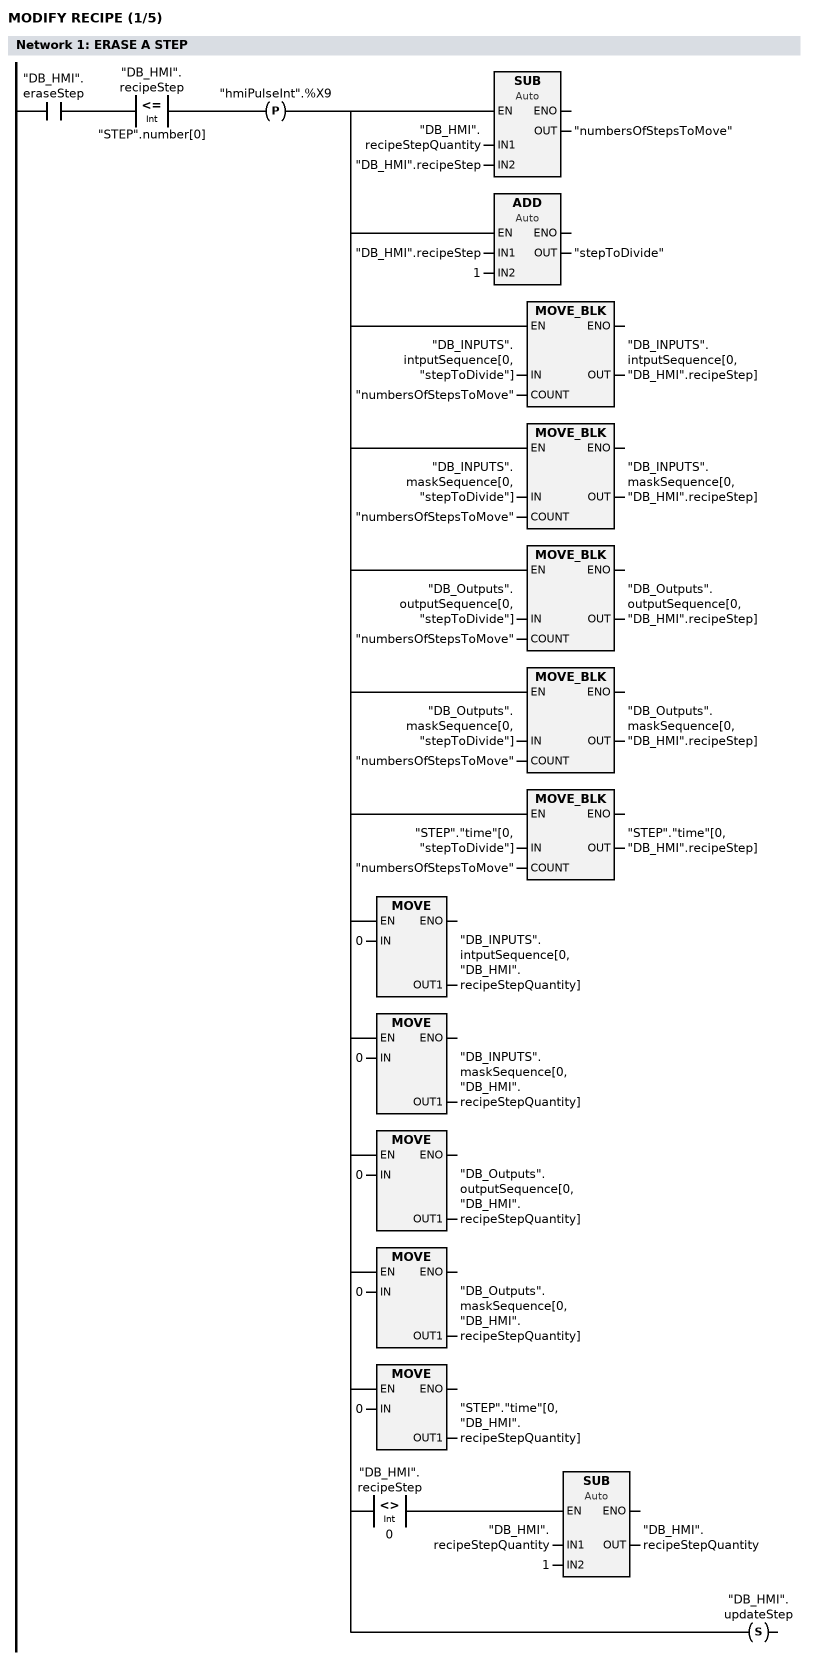
   #_w1 := "DB_HMI".eraseStep AND ("DB_HMI".recipeStep <= "STEP".number[0]);
   #_w2 := #_w1 AND NOT "hmiPulseInt".%X9;   // rising edge
   "hmiPulseInt".%X9 := #_w1;
   IF #_w2 THEN
       "numbersOfStepsToMove" := "DB_HMI".recipeStepQuantity - "DB_HMI".recipeStep;
       "stepToDivide" := "DB_HMI".recipeStep + 1;
       MOVE_BLK(IN := "DB_INPUTS".intputSequence[0, "stepToDivide"],
                COUNT := "numbersOfStepsToMove",
                OUT => "DB_INPUTS".intputSequence[0, "DB_HMI".recipeStep]);
       MOVE_BLK(IN := "DB_INPUTS".maskSequence[0, "stepToDivide"],
                COUNT := "numbersOfStepsToMove",
                OUT => "DB_INPUTS".maskSequence[0, "DB_HMI".recipeStep]);
       MOVE_BLK(IN := "DB_Outputs".outputSequence[0, "stepToDivide"],
                COUNT := "numbersOfStepsToMove",
                OUT => "DB_Outputs".outputSequence[0, "DB_HMI".recipeStep]);
       MOVE_BLK(IN := "DB_Outputs".maskSequence[0, "stepToDivide"],
                COUNT := "numbersOfStepsToMove",
                OUT => "DB_Outputs".maskSequence[0, "DB_HMI".recipeStep]);
       MOVE_BLK(IN := "STEP"."time"[0, "stepToDivide"],
                COUNT := "numbersOfStepsToMove",
                OUT => "STEP"."time"[0, "DB_HMI".recipeStep]);
       "DB_INPUTS".intputSequence[0, "DB_HMI".recipeStepQuantity] := 0;
       "DB_INPUTS".maskSequence[0, "DB_HMI".recipeStepQuantity] := 0;
       "DB_Outputs".outputSequence[0, "DB_HMI".recipeStepQuantity] := 0;
       "DB_Outputs".maskSequence[0, "DB_HMI".recipeStepQuantity] := 0;
       "STEP"."time"[0, "DB_HMI".recipeStepQuantity] := 0;
   END_IF;
   IF #_w2 AND ("DB_HMI".recipeStep <> 0) THEN
       "DB_HMI".recipeStepQuantity := "DB_HMI".recipeStepQuantity - 1;
   END_IF;
   IF #_w2 THEN "DB_HMI".updateStep := TRUE; END_IF;
END_REGION

REGION Network 2: ADD A STEP
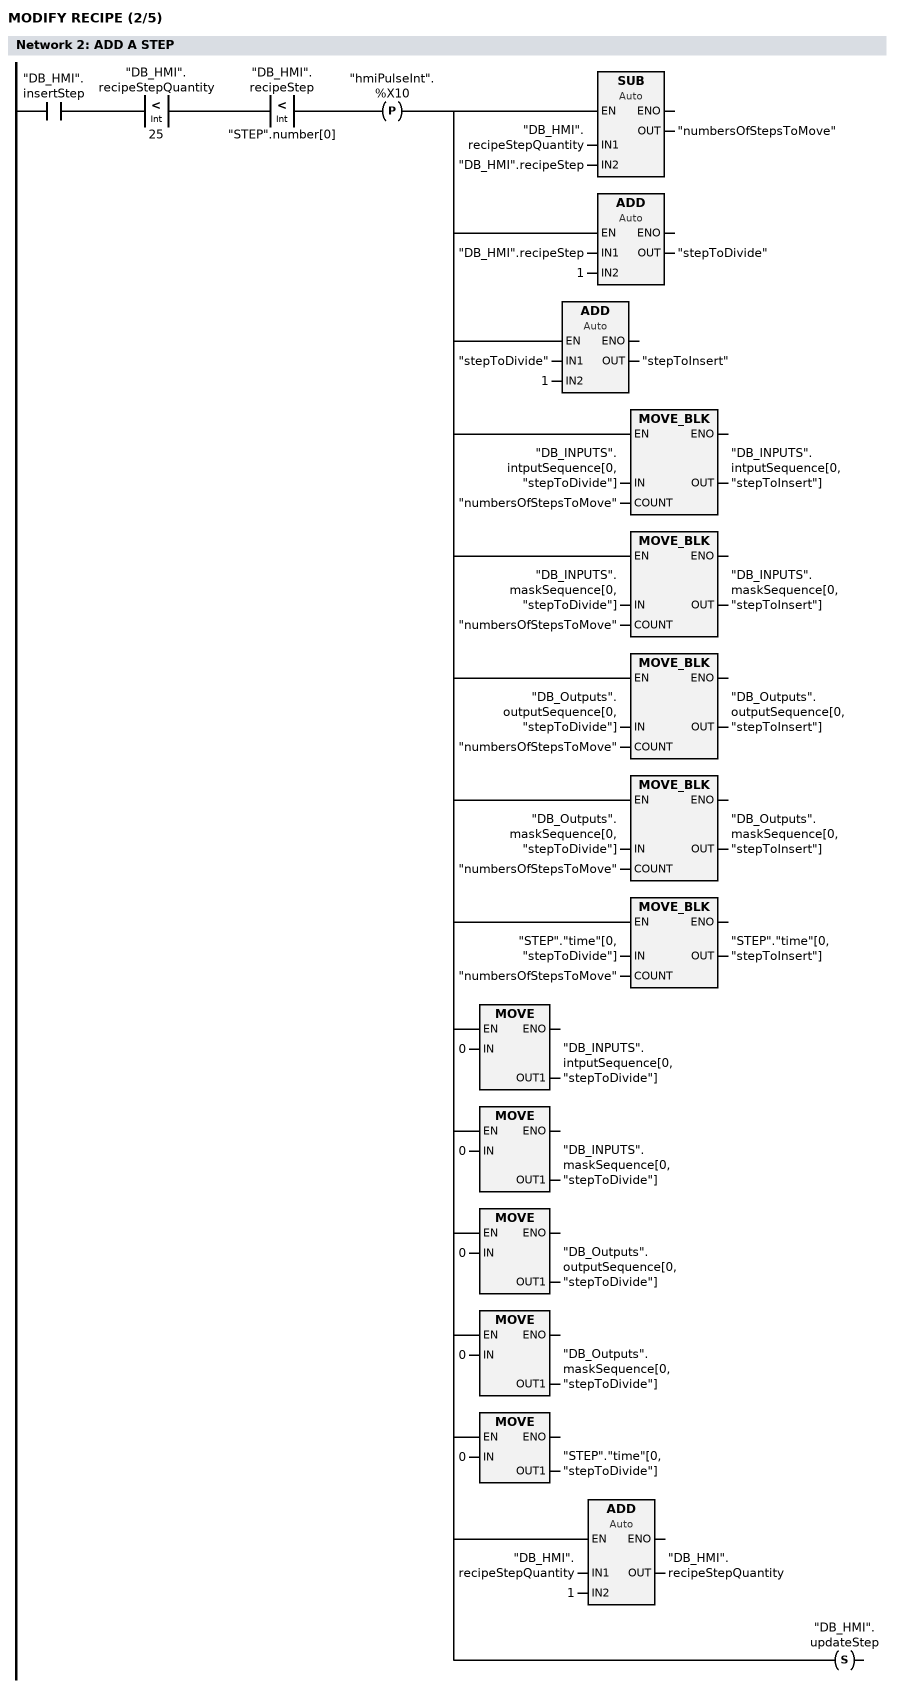
   #_w1 := "DB_HMI".insertStep AND ("DB_HMI".recipeStepQuantity < 25) AND ("DB_HMI".recipeStep < "STEP".number[0]);
   #_w2 := #_w1 AND NOT "hmiPulseInt".%X10;   // rising edge
   "hmiPulseInt".%X10 := #_w1;
   IF #_w2 THEN
       "numbersOfStepsToMove" := "DB_HMI".recipeStepQuantity - "DB_HMI".recipeStep;
       "stepToDivide" := "DB_HMI".recipeStep + 1;
       "stepToInsert" := "stepToDivide" + 1;
       MOVE_BLK(IN := "DB_INPUTS".intputSequence[0, "stepToDivide"],
                COUNT := "numbersOfStepsToMove",
                OUT => "DB_INPUTS".intputSequence[0, "stepToInsert"]);
       MOVE_BLK(IN := "DB_INPUTS".maskSequence[0, "stepToDivide"],
                COUNT := "numbersOfStepsToMove",
                OUT => "DB_INPUTS".maskSequence[0, "stepToInsert"]);
       MOVE_BLK(IN := "DB_Outputs".outputSequence[0, "stepToDivide"],
                COUNT := "numbersOfStepsToMove",
                OUT => "DB_Outputs".outputSequence[0, "stepToInsert"]);
       MOVE_BLK(IN := "DB_Outputs".maskSequence[0, "stepToDivide"],
                COUNT := "numbersOfStepsToMove",
                OUT => "DB_Outputs".maskSequence[0, "stepToInsert"]);
       MOVE_BLK(IN := "STEP"."time"[0, "stepToDivide"],
                COUNT := "numbersOfStepsToMove",
                OUT => "STEP"."time"[0, "stepToInsert"]);
       "DB_INPUTS".intputSequence[0, "stepToDivide"] := 0;
       "DB_INPUTS".maskSequence[0, "stepToDivide"] := 0;
       "DB_Outputs".outputSequence[0, "stepToDivide"] := 0;
       "DB_Outputs".maskSequence[0, "stepToDivide"] := 0;
       "STEP"."time"[0, "stepToDivide"] := 0;
       "DB_HMI".recipeStepQuantity := "DB_HMI".recipeStepQuantity + 1;
       "DB_HMI".updateStep := TRUE;
   END_IF;
END_REGION

REGION Network 3: COPY A STEP
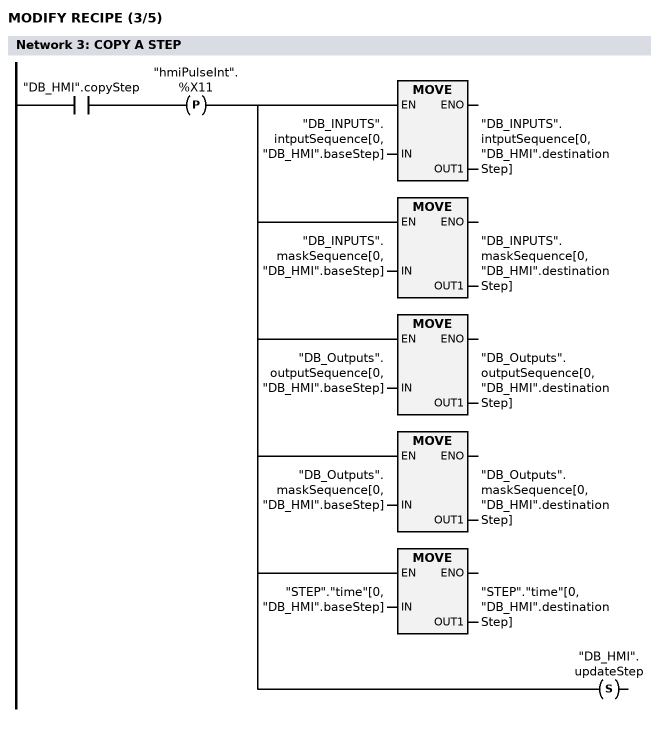
   RUNG wire#powerrail
      Contact( "DB_HMI".copyStep )
      P_Trig( "hmiPulseInt".%X11 )
      wire#w1
      Move(in := "DB_INPUTS".intputSequence[0, "DB_HMI".baseStep], out1 => "DB_INPUTS".intputSequence[0, "DB_HMI".destinationStep])
   END_RUNG
   RUNG wire#w1
      Move(in := "DB_INPUTS".maskSequence[0, "DB_HMI".baseStep], out1 => "DB_INPUTS".maskSequence[0, "DB_HMI".destinationStep])
   END_RUNG
   RUNG wire#w1
      Move(in := "DB_Outputs".outputSequence[0, "DB_HMI".baseStep], out1 => "DB_Outputs".outputSequence[0, "DB_HMI".destinationStep])
   END_RUNG
   RUNG wire#w1
      Move(in := "DB_Outputs".maskSequence[0, "DB_HMI".baseStep], out1 => "DB_Outputs".maskSequence[0, "DB_HMI".destinationStep])
   END_RUNG
   RUNG wire#w1
      Move(in := "STEP"."time"[0, "DB_HMI".baseStep], out1 => "STEP"."time"[0, "DB_HMI".destinationStep])
   END_RUNG
   RUNG wire#w1
      S_Coil( "DB_HMI".updateStep )
   END_RUNG
   // the same network as SCL:
   #_w1 := "DB_HMI".copyStep AND NOT "hmiPulseInt".%X11;   // rising edge
   "hmiPulseInt".%X11 := "DB_HMI".copyStep;
   IF #_w1 THEN
       "DB_INPUTS".intputSequence[0, "DB_HMI".destinationStep] := "DB_INPUTS".intputSequence[0, "DB_HMI".baseStep];
       "DB_INPUTS".maskSequence[0, "DB_HMI".destinationStep] := "DB_INPUTS".maskSequence[0, "DB_HMI".baseStep];
       "DB_Outputs".outputSequence[0, "DB_HMI".destinationStep] := "DB_Outputs".outputSequence[0, "DB_HMI".baseStep];
       "DB_Outputs".maskSequence[0, "DB_HMI".destinationStep] := "DB_Outputs".maskSequence[0, "DB_HMI".baseStep];
       "STEP"."time"[0, "DB_HMI".destinationStep] := "STEP"."time"[0, "DB_HMI".baseStep];
       "DB_HMI".updateStep := TRUE;
   END_IF;
END_REGION

REGION Network 4: COPY SEQUENCE (COPY PART NUMBER)
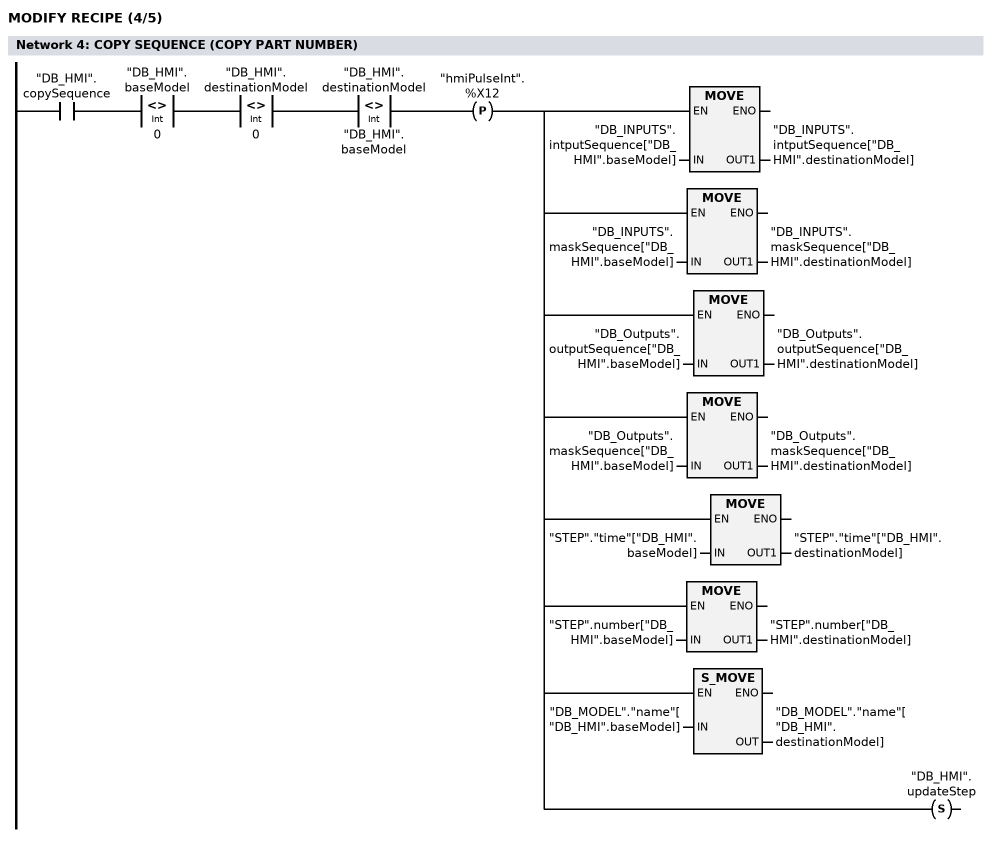
   RUNG wire#powerrail
      Contact( "DB_HMI".copySequence )
      { S7_Templates := "SrcType := Int" } NE_Contact(in1 := "DB_HMI".baseModel, in2 := 0)
      { S7_Templates := "SrcType := Int" } NE_Contact(in1 := "DB_HMI".destinationModel, in2 := 0)
      { S7_Templates := "SrcType := Int" } NE_Contact(in1 := "DB_HMI".destinationModel, in2 := "DB_HMI".baseModel)
      P_Trig( "hmiPulseInt".%X12 )
      wire#w1
      Move(in := "DB_INPUTS".intputSequence["DB_HMI".baseModel], out1 => "DB_INPUTS".intputSequence["DB_HMI".destinationModel])
   END_RUNG
   RUNG wire#w1
      Move(in := "DB_INPUTS".maskSequence["DB_HMI".baseModel], out1 => "DB_INPUTS".maskSequence["DB_HMI".destinationModel])
   END_RUNG
   RUNG wire#w1
      Move(in := "DB_Outputs".outputSequence["DB_HMI".baseModel], out1 => "DB_Outputs".outputSequence["DB_HMI".destinationModel])
   END_RUNG
   RUNG wire#w1
      Move(in := "DB_Outputs".maskSequence["DB_HMI".baseModel], out1 => "DB_Outputs".maskSequence["DB_HMI".destinationModel])
   END_RUNG
   RUNG wire#w1
      Move(in := "STEP"."time"["DB_HMI".baseModel], out1 => "STEP"."time"["DB_HMI".destinationModel])
   END_RUNG
   RUNG wire#w1
      Move(in := "STEP".number["DB_HMI".baseModel], out1 => "STEP".number["DB_HMI".destinationModel])
   END_RUNG
   RUNG wire#w1
      S_Move(in := "DB_MODEL"."name"["DB_HMI".baseModel], out => "DB_MODEL"."name"["DB_HMI".destinationModel])
   END_RUNG
   RUNG wire#w1
      S_Coil( "DB_HMI".updateStep )
   END_RUNG
   // the same network as SCL:
   #_w1 := "DB_HMI".copySequence AND ("DB_HMI".baseModel <> 0) AND ("DB_HMI".destinationModel <> 0) AND ("DB_HMI".destinationModel <> "DB_HMI".baseModel);
   #_w2 := #_w1 AND NOT "hmiPulseInt".%X12;   // rising edge
   "hmiPulseInt".%X12 := #_w1;
   IF #_w2 THEN
       "DB_INPUTS".intputSequence["DB_HMI".destinationModel] := "DB_INPUTS".intputSequence["DB_HMI".baseModel];
       "DB_INPUTS".maskSequence["DB_HMI".destinationModel] := "DB_INPUTS".maskSequence["DB_HMI".baseModel];
       "DB_Outputs".outputSequence["DB_HMI".destinationModel] := "DB_Outputs".outputSequence["DB_HMI".baseModel];
       "DB_Outputs".maskSequence["DB_HMI".destinationModel] := "DB_Outputs".maskSequence["DB_HMI".baseModel];
       "STEP"."time"["DB_HMI".destinationModel] := "STEP"."time"["DB_HMI".baseModel];
       "STEP".number["DB_HMI".destinationModel] := "STEP".number["DB_HMI".baseModel];
       "DB_MODEL"."name"["DB_HMI".destinationModel] := "DB_MODEL"."name"["DB_HMI".baseModel];
       "DB_HMI".updateStep := TRUE;
   END_IF;
END_REGION

REGION Network 5: COPY A STEP (#) FROM A PROGRAM (#) IN ANOTHER STEP (#) FROM ANOTHER PROGRAM (#)
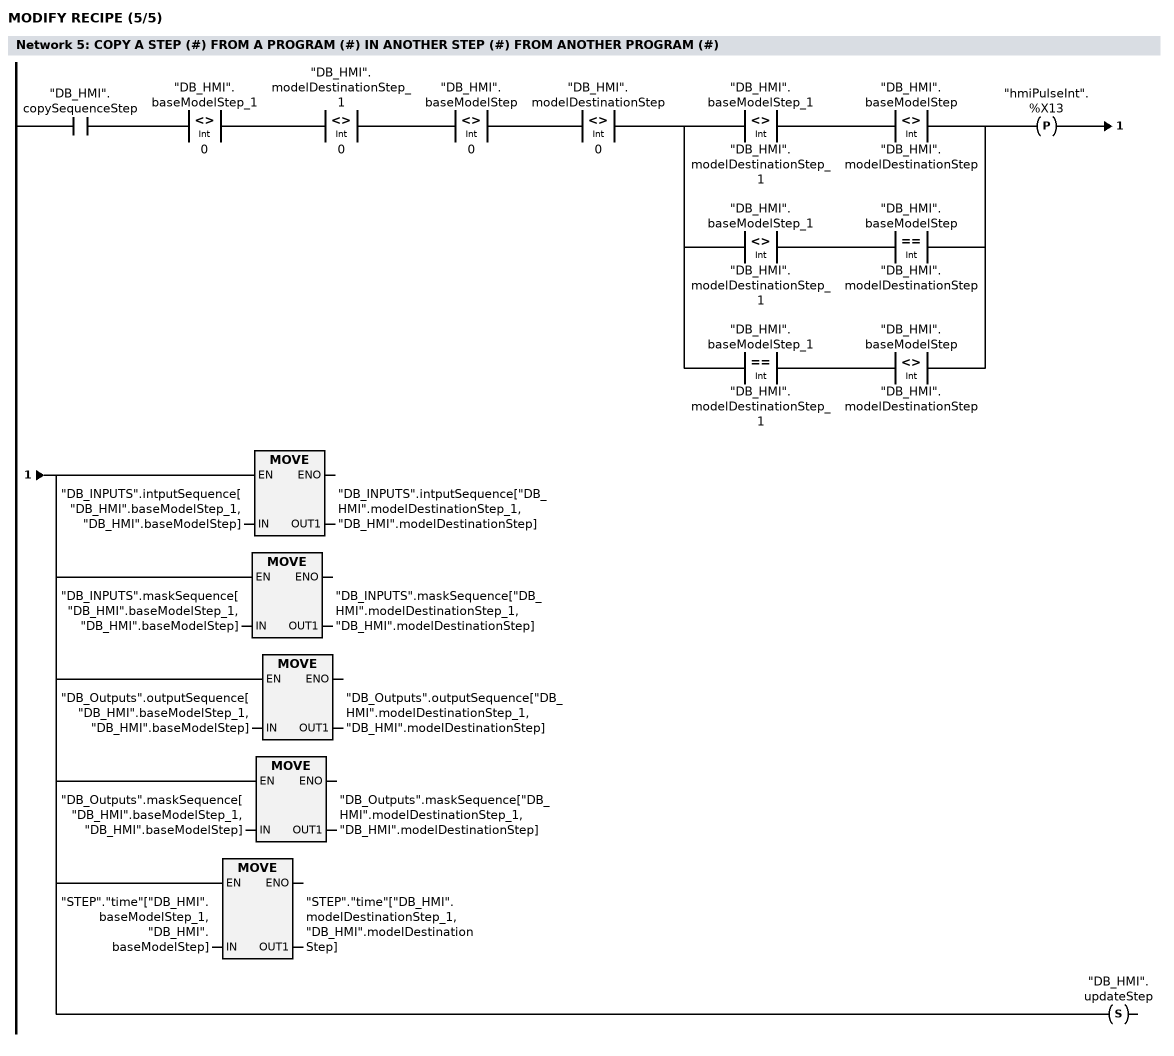
   RUNG wire#powerrail
      Contact( "DB_HMI".copySequenceStep )
      { S7_Templates := "SrcType := Int" } NE_Contact(in1 := "DB_HMI".baseModelStep_1, in2 := 0)
      { S7_Templates := "SrcType := Int" } NE_Contact(in1 := "DB_HMI".modelDestinationStep_1, in2 := 0)
      { S7_Templates := "SrcType := Int" } NE_Contact(in1 := "DB_HMI".baseModelStep, in2 := 0)
      { S7_Templates := "SrcType := Int" } NE_Contact(in1 := "DB_HMI".modelDestinationStep, in2 := 0)
      wire#w1
      { S7_Templates := "SrcType := Int" } NE_Contact(in1 := "DB_HMI".baseModelStep_1, in2 := "DB_HMI".modelDestinationStep_1)
      { S7_Templates := "SrcType := Int" } NE_Contact(in1 := "DB_HMI".baseModelStep, in2 := "DB_HMI".modelDestinationStep)
      wire#w2
      P_Trig( "hmiPulseInt".%X13 )
      wire#w3
      Move(in := "DB_INPUTS".intputSequence["DB_HMI".baseModelStep_1, "DB_HMI".baseModelStep], out1 => "DB_INPUTS".intputSequence["DB_HMI".modelDestinationStep_1, "DB_HMI".modelDestinationStep])
   END_RUNG
   RUNG wire#w1
      { S7_Templates := "SrcType := Int" } NE_Contact(in1 := "DB_HMI".baseModelStep_1, in2 := "DB_HMI".modelDestinationStep_1)
      { S7_Templates := "SrcType := Int" } EQ_Contact(in1 := "DB_HMI".baseModelStep, in2 := "DB_HMI".modelDestinationStep)
   END_RUNG wire#w2
   RUNG wire#w1
      { S7_Templates := "SrcType := Int" } EQ_Contact(in1 := "DB_HMI".baseModelStep_1, in2 := "DB_HMI".modelDestinationStep_1)
      { S7_Templates := "SrcType := Int" } NE_Contact(in1 := "DB_HMI".baseModelStep, in2 := "DB_HMI".modelDestinationStep)
   END_RUNG wire#w2
   RUNG wire#w3
      Move(in := "DB_INPUTS".maskSequence["DB_HMI".baseModelStep_1, "DB_HMI".baseModelStep], out1 => "DB_INPUTS".maskSequence["DB_HMI".modelDestinationStep_1, "DB_HMI".modelDestinationStep])
   END_RUNG
   RUNG wire#w3
      Move(in := "DB_Outputs".outputSequence["DB_HMI".baseModelStep_1, "DB_HMI".baseModelStep], out1 => "DB_Outputs".outputSequence["DB_HMI".modelDestinationStep_1, "DB_HMI".modelDestinationStep])
   END_RUNG
   RUNG wire#w3
      Move(in := "DB_Outputs".maskSequence["DB_HMI".baseModelStep_1, "DB_HMI".baseModelStep], out1 => "DB_Outputs".maskSequence["DB_HMI".modelDestinationStep_1, "DB_HMI".modelDestinationStep])
   END_RUNG
   RUNG wire#w3
      Move(in := "STEP"."time"["DB_HMI".baseModelStep_1, "DB_HMI".baseModelStep], out1 => "STEP"."time"["DB_HMI".modelDestinationStep_1, "DB_HMI".modelDestinationStep])
   END_RUNG
   RUNG wire#w3
      S_Coil( "DB_HMI".updateStep )
   END_RUNG
   // the same network as SCL:
   #_w1 := "DB_HMI".copySequenceStep AND ("DB_HMI".baseModelStep_1 <> 0) AND ("DB_HMI".modelDestinationStep_1 <> 0) AND ("DB_HMI".baseModelStep <> 0) AND ("DB_HMI".modelDestinationStep <> 0) AND ((("DB_HMI".baseModelStep_1 <> "DB_HMI".modelDestinationStep_1) AND ("DB_HMI".baseModelStep <> "DB_HMI".modelDestinationStep)) OR (("DB_HMI".baseModelStep_1 <> "DB_HMI".modelDestinationStep_1) AND ("DB_HMI".baseModelStep = "DB_HMI".modelDestinationStep)) OR (("DB_HMI".baseModelStep_1 = "DB_HMI".modelDestinationStep_1) AND ("DB_HMI".baseModelStep <> "DB_HMI".modelDestinationStep)));
   #_w2 := #_w1 AND NOT "hmiPulseInt".%X13;   // rising edge
   "hmiPulseInt".%X13 := #_w1;
   IF #_w2 THEN
       "DB_INPUTS".intputSequence["DB_HMI".modelDestinationStep_1, "DB_HMI".modelDestinationStep] := "DB_INPUTS".intputSequence["DB_HMI".baseModelStep_1, "DB_HMI".baseModelStep];
       "DB_INPUTS".maskSequence["DB_HMI".modelDestinationStep_1, "DB_HMI".modelDestinationStep] := "DB_INPUTS".maskSequence["DB_HMI".baseModelStep_1, "DB_HMI".baseModelStep];
       "DB_Outputs".outputSequence["DB_HMI".modelDestinationStep_1, "DB_HMI".modelDestinationStep] := "DB_Outputs".outputSequence["DB_HMI".baseModelStep_1, "DB_HMI".baseModelStep];
       "DB_Outputs".maskSequence["DB_HMI".modelDestinationStep_1, "DB_HMI".modelDestinationStep] := "DB_Outputs".maskSequence["DB_HMI".baseModelStep_1, "DB_HMI".baseModelStep];
       "STEP"."time"["DB_HMI".modelDestinationStep_1, "DB_HMI".modelDestinationStep] := "STEP"."time"["DB_HMI".baseModelStep_1, "DB_HMI".baseModelStep];
       "DB_HMI".updateStep := TRUE;
   END_IF;
END_REGION
END_FUNCTION

FUNCTION "inputsMapping" : Void   // FC1, LAD
{ S7_Optimized_Access := 'TRUE' }
VERSION : 0.1
// stored: AutoNumber true, IsIECCheckEnabled false, SetENOAutomatically false, UDAEnableTagReadback false
BEGIN

REGION Network 1: A00.- CLEAR DATA
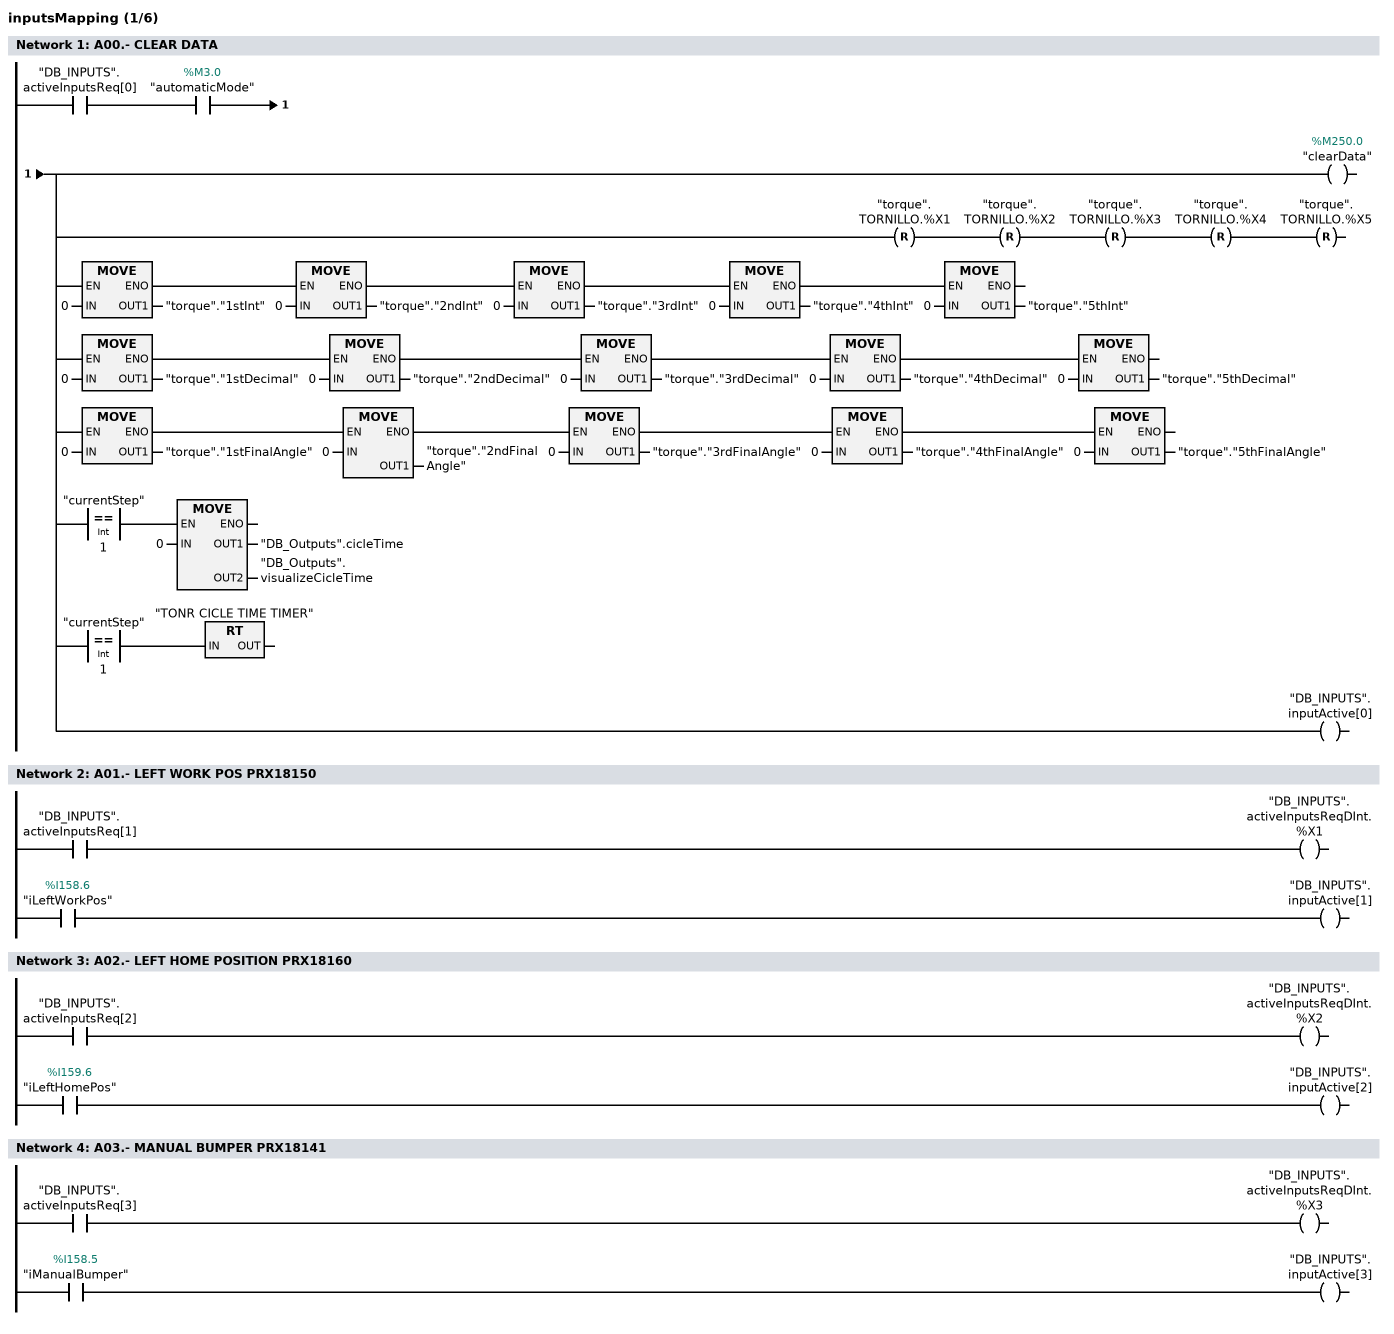
   RUNG wire#powerrail
      Contact( "DB_INPUTS".activeInputsReq[0] )
      Contact( "automaticMode" )
      wire#w1
      Coil( "clearData" )
   END_RUNG
   RUNG wire#w1
      R_Coil( "torque".TORNILLO.%X1 )
      R_Coil( "torque".TORNILLO.%X2 )
      R_Coil( "torque".TORNILLO.%X3 )
      R_Coil( "torque".TORNILLO.%X4 )
      R_Coil( "torque".TORNILLO.%X5 )
   END_RUNG
   RUNG wire#w1
      Move(in := 0, out1 => "torque"."1stInt")
      Move(in := 0, out1 => "torque"."2ndInt")
      Move(in := 0, out1 => "torque"."3rdInt")
      Move(in := 0, out1 => "torque"."4thInt")
      Move(in := 0, out1 => "torque"."5thInt")
   END_RUNG
   RUNG wire#w1
      Move(in := 0, out1 => "torque"."1stDecimal")
      Move(in := 0, out1 => "torque"."2ndDecimal")
      Move(in := 0, out1 => "torque"."3rdDecimal")
      Move(in := 0, out1 => "torque"."4thDecimal")
      Move(in := 0, out1 => "torque"."5thDecimal")
   END_RUNG
   RUNG wire#w1
      Move(in := 0, out1 => "torque"."1stFinalAngle")
      Move(in := 0, out1 => "torque"."2ndFinalAngle")
      Move(in := 0, out1 => "torque"."3rdFinalAngle")
      Move(in := 0, out1 => "torque"."4thFinalAngle")
      Move(in := 0, out1 => "torque"."5thFinalAngle")
   END_RUNG
   RUNG wire#w1
      { S7_Templates := "SrcType := Int" } EQ_Contact(in1 := "currentStep", in2 := 1)
      Move(in := 0, out1 => "DB_Outputs".cicleTime, out2 => "DB_Outputs".visualizeCicleTime)
   END_RUNG
   RUNG wire#w1
      { S7_Templates := "SrcType := Int" } EQ_Contact(in1 := "currentStep", in2 := 1)
      RT_Coil( "TONR CICLE TIME TIMER" )
   END_RUNG
   RUNG wire#w1
      Coil( "DB_INPUTS".inputActive[0] )
   END_RUNG
   // the same network as SCL:
   "clearData" := "DB_INPUTS".activeInputsReq[0] AND "automaticMode";
   IF "clearData" THEN
       "torque".TORNILLO.%X1 := FALSE;
       "torque".TORNILLO.%X2 := FALSE;
       "torque".TORNILLO.%X3 := FALSE;
       "torque".TORNILLO.%X4 := FALSE;
       "torque".TORNILLO.%X5 := FALSE;
       "torque"."1stInt" := 0;
       "torque"."2ndInt" := 0;
       "torque"."3rdInt" := 0;
       "torque"."4thInt" := 0;
       "torque"."5thInt" := 0;
       "torque"."1stDecimal" := 0;
       "torque"."2ndDecimal" := 0;
       "torque"."3rdDecimal" := 0;
       "torque"."4thDecimal" := 0;
       "torque"."5thDecimal" := 0;
       "torque"."1stFinalAngle" := 0;
       "torque"."2ndFinalAngle" := 0;
       "torque"."3rdFinalAngle" := 0;
       "torque"."4thFinalAngle" := 0;
       "torque"."5thFinalAngle" := 0;
   END_IF;
   IF "clearData" AND ("currentStep" = 1) THEN
       "DB_Outputs".cicleTime := 0;
       "DB_Outputs".visualizeCicleTime := 0;
       RESET_TIMER("TONR CICLE TIME TIMER");
   END_IF;
   "DB_INPUTS".inputActive[0] := "clearData";
END_REGION

REGION Network 2: A01.- LEFT WORK POS PRX18150
   RUNG wire#powerrail
      Contact( "DB_INPUTS".activeInputsReq[1] )
      Coil( "DB_INPUTS".activeInputsReqDInt.%X1 )
   END_RUNG
   RUNG wire#powerrail
      Contact( "iLeftWorkPos" )
      Coil( "DB_INPUTS".inputActive[1] )
   END_RUNG
   // the same network as SCL:
   "DB_INPUTS".activeInputsReqDInt.%X1 := "DB_INPUTS".activeInputsReq[1];
   "DB_INPUTS".inputActive[1] := "iLeftWorkPos";
END_REGION

REGION Network 3: A02.- LEFT HOME POSITION PRX18160
   RUNG wire#powerrail
      Contact( "DB_INPUTS".activeInputsReq[2] )
      Coil( "DB_INPUTS".activeInputsReqDInt.%X2 )
   END_RUNG
   RUNG wire#powerrail
      Contact( "iLeftHomePos" )
      Coil( "DB_INPUTS".inputActive[2] )
   END_RUNG
   // the same network as SCL:
   "DB_INPUTS".activeInputsReqDInt.%X2 := "DB_INPUTS".activeInputsReq[2];
   "DB_INPUTS".inputActive[2] := "iLeftHomePos";
END_REGION

REGION Network 4: A03.- MANUAL BUMPER PRX18141
   RUNG wire#powerrail
      Contact( "DB_INPUTS".activeInputsReq[3] )
      Coil( "DB_INPUTS".activeInputsReqDInt.%X3 )
   END_RUNG
   RUNG wire#powerrail
      Contact( "iManualBumper" )
      Coil( "DB_INPUTS".inputActive[3] )
   END_RUNG
   // the same network as SCL:
   "DB_INPUTS".activeInputsReqDInt.%X3 := "DB_INPUTS".activeInputsReq[3];
   "DB_INPUTS".inputActive[3] := "iManualBumper";
END_REGION

REGION Network 5: A04.- LEFT MANUAL TOOLING EXT OK PRX18151
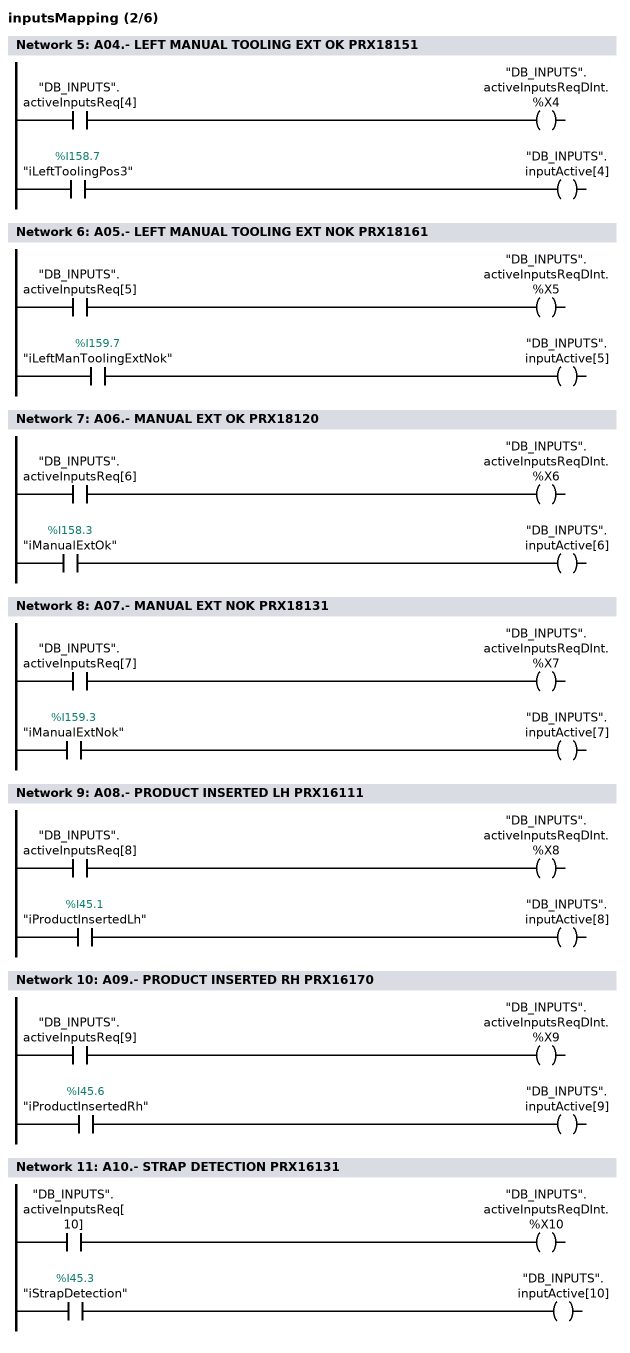
   RUNG wire#powerrail
      Contact( "DB_INPUTS".activeInputsReq[4] )
      Coil( "DB_INPUTS".activeInputsReqDInt.%X4 )
   END_RUNG
   RUNG wire#powerrail
      Contact( "iLeftToolingPos3" )
      Coil( "DB_INPUTS".inputActive[4] )
   END_RUNG
   // the same network as SCL:
   "DB_INPUTS".activeInputsReqDInt.%X4 := "DB_INPUTS".activeInputsReq[4];
   "DB_INPUTS".inputActive[4] := "iLeftToolingPos3";
END_REGION

REGION Network 6: A05.- LEFT MANUAL TOOLING EXT NOK PRX18161
   RUNG wire#powerrail
      Contact( "DB_INPUTS".activeInputsReq[5] )
      Coil( "DB_INPUTS".activeInputsReqDInt.%X5 )
   END_RUNG
   RUNG wire#powerrail
      Contact( "iLeftManToolingExtNok" )
      Coil( "DB_INPUTS".inputActive[5] )
   END_RUNG
   // the same network as SCL:
   "DB_INPUTS".activeInputsReqDInt.%X5 := "DB_INPUTS".activeInputsReq[5];
   "DB_INPUTS".inputActive[5] := "iLeftManToolingExtNok";
END_REGION

REGION Network 7: A06.- MANUAL EXT OK PRX18120
   RUNG wire#powerrail
      Contact( "DB_INPUTS".activeInputsReq[6] )
      Coil( "DB_INPUTS".activeInputsReqDInt.%X6 )
   END_RUNG
   RUNG wire#powerrail
      Contact( "iManualExtOk" )
      Coil( "DB_INPUTS".inputActive[6] )
   END_RUNG
   // the same network as SCL:
   "DB_INPUTS".activeInputsReqDInt.%X6 := "DB_INPUTS".activeInputsReq[6];
   "DB_INPUTS".inputActive[6] := "iManualExtOk";
END_REGION

REGION Network 8: A07.- MANUAL EXT NOK PRX18131
   RUNG wire#powerrail
      Contact( "DB_INPUTS".activeInputsReq[7] )
      Coil( "DB_INPUTS".activeInputsReqDInt.%X7 )
   END_RUNG
   RUNG wire#powerrail
      Contact( "iManualExtNok" )
      Coil( "DB_INPUTS".inputActive[7] )
   END_RUNG
   // the same network as SCL:
   "DB_INPUTS".activeInputsReqDInt.%X7 := "DB_INPUTS".activeInputsReq[7];
   "DB_INPUTS".inputActive[7] := "iManualExtNok";
END_REGION

REGION Network 9: A08.- PRODUCT INSERTED LH PRX16111
   RUNG wire#powerrail
      Contact( "DB_INPUTS".activeInputsReq[8] )
      Coil( "DB_INPUTS".activeInputsReqDInt.%X8 )
   END_RUNG
   RUNG wire#powerrail
      Contact( "iProductInsertedLh" )
      Coil( "DB_INPUTS".inputActive[8] )
   END_RUNG
   // the same network as SCL:
   "DB_INPUTS".activeInputsReqDInt.%X8 := "DB_INPUTS".activeInputsReq[8];
   "DB_INPUTS".inputActive[8] := "iProductInsertedLh";
END_REGION

REGION Network 10: A09.- PRODUCT INSERTED RH PRX16170
   RUNG wire#powerrail
      Contact( "DB_INPUTS".activeInputsReq[9] )
      Coil( "DB_INPUTS".activeInputsReqDInt.%X9 )
   END_RUNG
   RUNG wire#powerrail
      Contact( "iProductInsertedRh" )
      Coil( "DB_INPUTS".inputActive[9] )
   END_RUNG
   // the same network as SCL:
   "DB_INPUTS".activeInputsReqDInt.%X9 := "DB_INPUTS".activeInputsReq[9];
   "DB_INPUTS".inputActive[9] := "iProductInsertedRh";
END_REGION

REGION Network 11: A10.- STRAP DETECTION PRX16131
   RUNG wire#powerrail
      Contact( "DB_INPUTS".activeInputsReq[10] )
      Coil( "DB_INPUTS".activeInputsReqDInt.%X10 )
   END_RUNG
   RUNG wire#powerrail
      Contact( "iStrapDetection" )
      Coil( "DB_INPUTS".inputActive[10] )
   END_RUNG
   // the same network as SCL:
   "DB_INPUTS".activeInputsReqDInt.%X10 := "DB_INPUTS".activeInputsReq[10];
   "DB_INPUTS".inputActive[10] := "iStrapDetection";
END_REGION

REGION Network 12: A11.- PRESENT LEFT MANUAL FRAME PRX17111
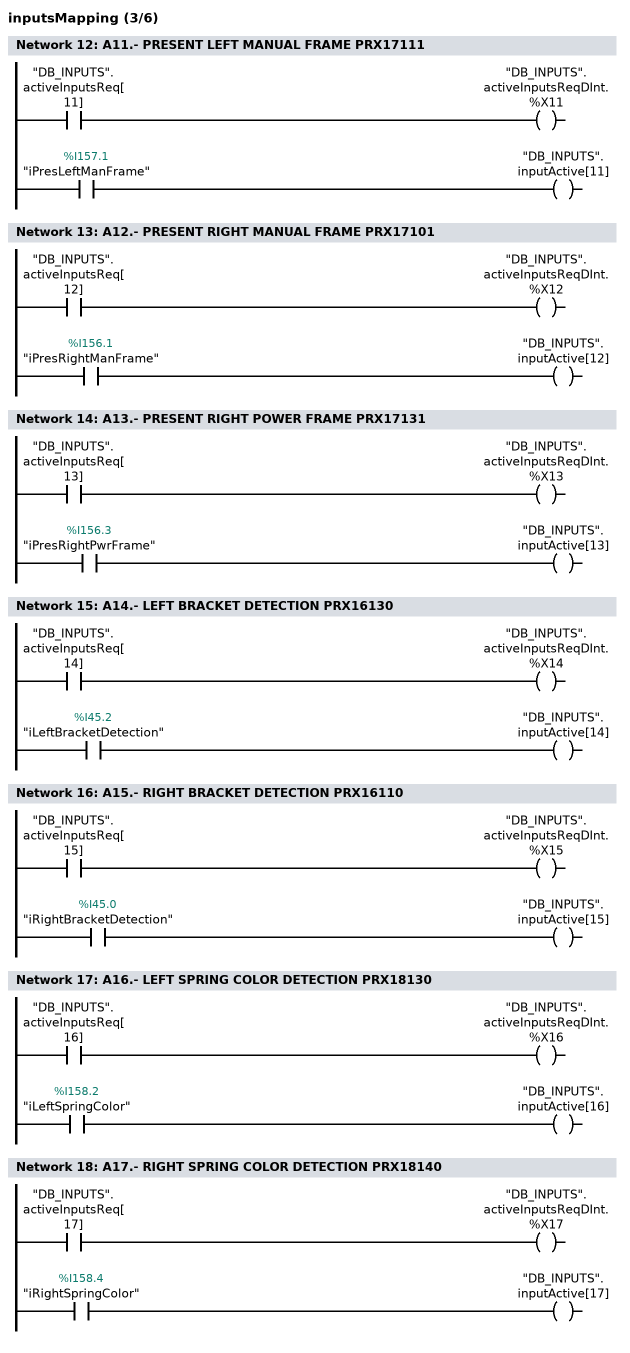
   RUNG wire#powerrail
      Contact( "DB_INPUTS".activeInputsReq[11] )
      Coil( "DB_INPUTS".activeInputsReqDInt.%X11 )
   END_RUNG
   RUNG wire#powerrail
      Contact( "iPresLeftManFrame" )
      Coil( "DB_INPUTS".inputActive[11] )
   END_RUNG
   // the same network as SCL:
   "DB_INPUTS".activeInputsReqDInt.%X11 := "DB_INPUTS".activeInputsReq[11];
   "DB_INPUTS".inputActive[11] := "iPresLeftManFrame";
END_REGION

REGION Network 13: A12.- PRESENT RIGHT MANUAL FRAME PRX17101
   RUNG wire#powerrail
      Contact( "DB_INPUTS".activeInputsReq[12] )
      Coil( "DB_INPUTS".activeInputsReqDInt.%X12 )
   END_RUNG
   RUNG wire#powerrail
      Contact( "iPresRightManFrame" )
      Coil( "DB_INPUTS".inputActive[12] )
   END_RUNG
   // the same network as SCL:
   "DB_INPUTS".activeInputsReqDInt.%X12 := "DB_INPUTS".activeInputsReq[12];
   "DB_INPUTS".inputActive[12] := "iPresRightManFrame";
END_REGION

REGION Network 14: A13.- PRESENT RIGHT POWER FRAME PRX17131
   RUNG wire#powerrail
      Contact( "DB_INPUTS".activeInputsReq[13] )
      Coil( "DB_INPUTS".activeInputsReqDInt.%X13 )
   END_RUNG
   RUNG wire#powerrail
      Contact( "iPresRightPwrFrame" )
      Coil( "DB_INPUTS".inputActive[13] )
   END_RUNG
   // the same network as SCL:
   "DB_INPUTS".activeInputsReqDInt.%X13 := "DB_INPUTS".activeInputsReq[13];
   "DB_INPUTS".inputActive[13] := "iPresRightPwrFrame";
END_REGION

REGION Network 15: A14.- LEFT BRACKET DETECTION PRX16130
   RUNG wire#powerrail
      Contact( "DB_INPUTS".activeInputsReq[14] )
      Coil( "DB_INPUTS".activeInputsReqDInt.%X14 )
   END_RUNG
   RUNG wire#powerrail
      Contact( "iLeftBracketDetection" )
      Coil( "DB_INPUTS".inputActive[14] )
   END_RUNG
   // the same network as SCL:
   "DB_INPUTS".activeInputsReqDInt.%X14 := "DB_INPUTS".activeInputsReq[14];
   "DB_INPUTS".inputActive[14] := "iLeftBracketDetection";
END_REGION

REGION Network 16: A15.- RIGHT BRACKET DETECTION PRX16110
   RUNG wire#powerrail
      Contact( "DB_INPUTS".activeInputsReq[15] )
      Coil( "DB_INPUTS".activeInputsReqDInt.%X15 )
   END_RUNG
   RUNG wire#powerrail
      Contact( "iRightBracketDetection" )
      Coil( "DB_INPUTS".inputActive[15] )
   END_RUNG
   // the same network as SCL:
   "DB_INPUTS".activeInputsReqDInt.%X15 := "DB_INPUTS".activeInputsReq[15];
   "DB_INPUTS".inputActive[15] := "iRightBracketDetection";
END_REGION

REGION Network 17: A16.- LEFT SPRING COLOR DETECTION PRX18130
   RUNG wire#powerrail
      Contact( "DB_INPUTS".activeInputsReq[16] )
      Coil( "DB_INPUTS".activeInputsReqDInt.%X16 )
   END_RUNG
   RUNG wire#powerrail
      Contact( "iLeftSpringColor" )
      Coil( "DB_INPUTS".inputActive[16] )
   END_RUNG
   // the same network as SCL:
   "DB_INPUTS".activeInputsReqDInt.%X16 := "DB_INPUTS".activeInputsReq[16];
   "DB_INPUTS".inputActive[16] := "iLeftSpringColor";
END_REGION

REGION Network 18: A17.- RIGHT SPRING COLOR DETECTION PRX18140
   RUNG wire#powerrail
      Contact( "DB_INPUTS".activeInputsReq[17] )
      Coil( "DB_INPUTS".activeInputsReqDInt.%X17 )
   END_RUNG
   RUNG wire#powerrail
      Contact( "iRightSpringColor" )
      Coil( "DB_INPUTS".inputActive[17] )
   END_RUNG
   // the same network as SCL:
   "DB_INPUTS".activeInputsReqDInt.%X17 := "DB_INPUTS".activeInputsReq[17];
   "DB_INPUTS".inputActive[17] := "iRightSpringColor";
END_REGION

REGION Network 19: A18.- TORQUE TOOLING HOME PRX16151
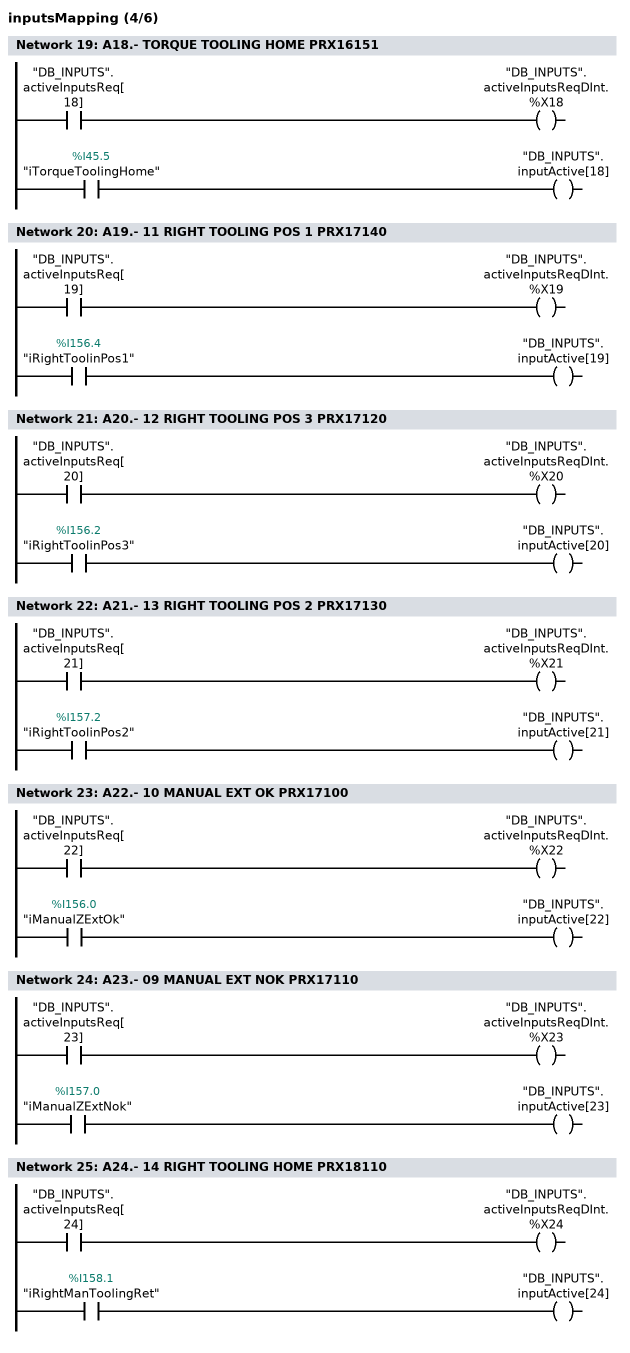
   RUNG wire#powerrail
      Contact( "DB_INPUTS".activeInputsReq[18] )
      Coil( "DB_INPUTS".activeInputsReqDInt.%X18 )
   END_RUNG
   RUNG wire#powerrail
      Contact( "iTorqueToolingHome" )
      Coil( "DB_INPUTS".inputActive[18] )
   END_RUNG
   // the same network as SCL:
   "DB_INPUTS".activeInputsReqDInt.%X18 := "DB_INPUTS".activeInputsReq[18];
   "DB_INPUTS".inputActive[18] := "iTorqueToolingHome";
END_REGION

REGION Network 20: A19.- 11 RIGHT TOOLING POS 1 PRX17140
   RUNG wire#powerrail
      Contact( "DB_INPUTS".activeInputsReq[19] )
      Coil( "DB_INPUTS".activeInputsReqDInt.%X19 )
   END_RUNG
   RUNG wire#powerrail
      Contact( "iRightToolinPos1" )
      Coil( "DB_INPUTS".inputActive[19] )
   END_RUNG
   // the same network as SCL:
   "DB_INPUTS".activeInputsReqDInt.%X19 := "DB_INPUTS".activeInputsReq[19];
   "DB_INPUTS".inputActive[19] := "iRightToolinPos1";
END_REGION

REGION Network 21: A20.- 12 RIGHT TOOLING POS 3 PRX17120
   RUNG wire#powerrail
      Contact( "DB_INPUTS".activeInputsReq[20] )
      Coil( "DB_INPUTS".activeInputsReqDInt.%X20 )
   END_RUNG
   RUNG wire#powerrail
      Contact( "iRightToolinPos3" )
      Coil( "DB_INPUTS".inputActive[20] )
   END_RUNG
   // the same network as SCL:
   "DB_INPUTS".activeInputsReqDInt.%X20 := "DB_INPUTS".activeInputsReq[20];
   "DB_INPUTS".inputActive[20] := "iRightToolinPos3";
END_REGION

REGION Network 22: A21.- 13 RIGHT TOOLING POS 2 PRX17130
   RUNG wire#powerrail
      Contact( "DB_INPUTS".activeInputsReq[21] )
      Coil( "DB_INPUTS".activeInputsReqDInt.%X21 )
   END_RUNG
   RUNG wire#powerrail
      Contact( "iRightToolinPos2" )
      Coil( "DB_INPUTS".inputActive[21] )
   END_RUNG
   // the same network as SCL:
   "DB_INPUTS".activeInputsReqDInt.%X21 := "DB_INPUTS".activeInputsReq[21];
   "DB_INPUTS".inputActive[21] := "iRightToolinPos2";
END_REGION

REGION Network 23: A22.- 10 MANUAL EXT OK PRX17100
   RUNG wire#powerrail
      Contact( "DB_INPUTS".activeInputsReq[22] )
      Coil( "DB_INPUTS".activeInputsReqDInt.%X22 )
   END_RUNG
   RUNG wire#powerrail
      Contact( "iManualZExtOk" )
      Coil( "DB_INPUTS".inputActive[22] )
   END_RUNG
   // the same network as SCL:
   "DB_INPUTS".activeInputsReqDInt.%X22 := "DB_INPUTS".activeInputsReq[22];
   "DB_INPUTS".inputActive[22] := "iManualZExtOk";
END_REGION

REGION Network 24: A23.- 09 MANUAL EXT NOK PRX17110
   RUNG wire#powerrail
      Contact( "DB_INPUTS".activeInputsReq[23] )
      Coil( "DB_INPUTS".activeInputsReqDInt.%X23 )
   END_RUNG
   RUNG wire#powerrail
      Contact( "iManualZExtNok" )
      Coil( "DB_INPUTS".inputActive[23] )
   END_RUNG
   // the same network as SCL:
   "DB_INPUTS".activeInputsReqDInt.%X23 := "DB_INPUTS".activeInputsReq[23];
   "DB_INPUTS".inputActive[23] := "iManualZExtNok";
END_REGION

REGION Network 25: A24.- 14 RIGHT TOOLING HOME PRX18110
   RUNG wire#powerrail
      Contact( "DB_INPUTS".activeInputsReq[24] )
      Coil( "DB_INPUTS".activeInputsReqDInt.%X24 )
   END_RUNG
   RUNG wire#powerrail
      Contact( "iRightManToolingRet" )
      Coil( "DB_INPUTS".inputActive[24] )
   END_RUNG
   // the same network as SCL:
   "DB_INPUTS".activeInputsReqDInt.%X24 := "DB_INPUTS".activeInputsReq[24];
   "DB_INPUTS".inputActive[24] := "iRightManToolingRet";
END_REGION

REGION Network 26: A25.- WASHER PRESENCE
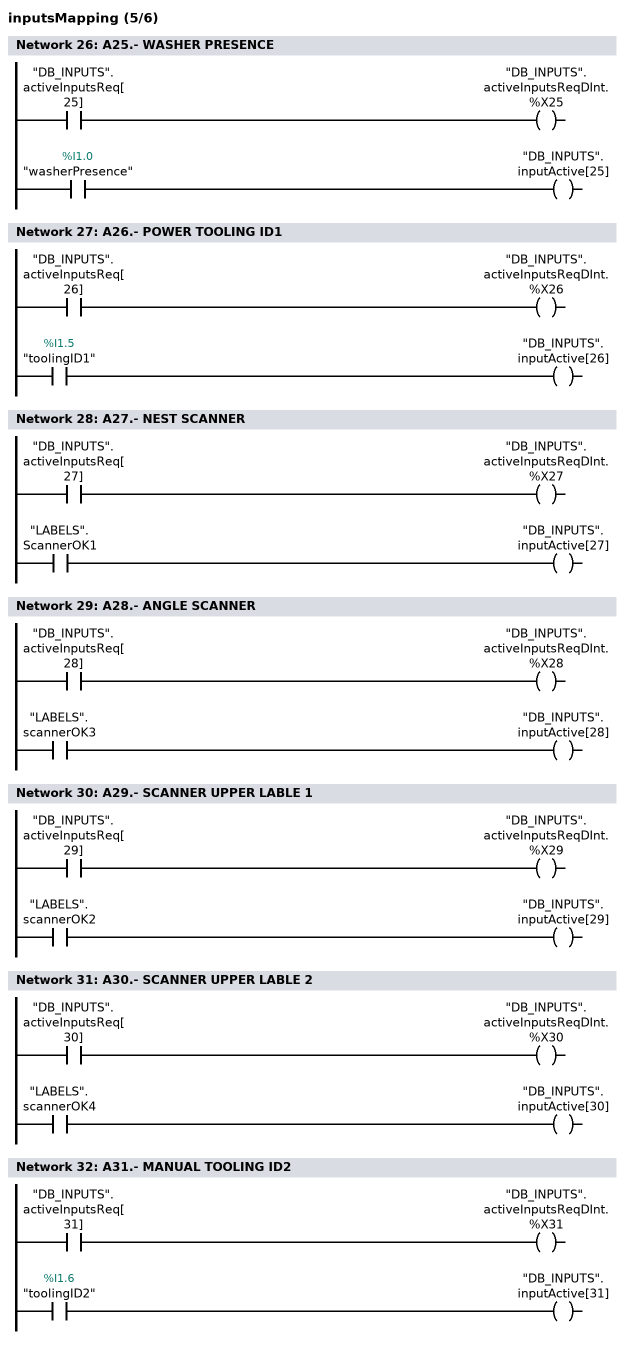
   RUNG wire#powerrail
      Contact( "DB_INPUTS".activeInputsReq[25] )
      Coil( "DB_INPUTS".activeInputsReqDInt.%X25 )
   END_RUNG
   RUNG wire#powerrail
      Contact( "washerPresence" )
      Coil( "DB_INPUTS".inputActive[25] )
   END_RUNG
   // the same network as SCL:
   "DB_INPUTS".activeInputsReqDInt.%X25 := "DB_INPUTS".activeInputsReq[25];
   "DB_INPUTS".inputActive[25] := "washerPresence";
END_REGION

REGION Network 27: A26.- POWER TOOLING ID1
   RUNG wire#powerrail
      Contact( "DB_INPUTS".activeInputsReq[26] )
      Coil( "DB_INPUTS".activeInputsReqDInt.%X26 )
   END_RUNG
   RUNG wire#powerrail
      Contact( "toolingID1" )
      Coil( "DB_INPUTS".inputActive[26] )
   END_RUNG
   // the same network as SCL:
   "DB_INPUTS".activeInputsReqDInt.%X26 := "DB_INPUTS".activeInputsReq[26];
   "DB_INPUTS".inputActive[26] := "toolingID1";
END_REGION

REGION Network 28: A27.- NEST SCANNER
   RUNG wire#powerrail
      Contact( "DB_INPUTS".activeInputsReq[27] )
      Coil( "DB_INPUTS".activeInputsReqDInt.%X27 )
   END_RUNG
   RUNG wire#powerrail
      Contact( "LABELS".ScannerOK1 )
      Coil( "DB_INPUTS".inputActive[27] )
   END_RUNG
   // the same network as SCL:
   "DB_INPUTS".activeInputsReqDInt.%X27 := "DB_INPUTS".activeInputsReq[27];
   "DB_INPUTS".inputActive[27] := "LABELS".ScannerOK1;
END_REGION

REGION Network 29: A28.- ANGLE SCANNER
   RUNG wire#powerrail
      Contact( "DB_INPUTS".activeInputsReq[28] )
      Coil( "DB_INPUTS".activeInputsReqDInt.%X28 )
   END_RUNG
   RUNG wire#powerrail
      Contact( "LABELS".scannerOK3 )
      Coil( "DB_INPUTS".inputActive[28] )
   END_RUNG
   // the same network as SCL:
   "DB_INPUTS".activeInputsReqDInt.%X28 := "DB_INPUTS".activeInputsReq[28];
   "DB_INPUTS".inputActive[28] := "LABELS".scannerOK3;
END_REGION

REGION Network 30: A29.- SCANNER UPPER LABLE 1
   RUNG wire#powerrail
      Contact( "DB_INPUTS".activeInputsReq[29] )
      Coil( "DB_INPUTS".activeInputsReqDInt.%X29 )
   END_RUNG
   RUNG wire#powerrail
      Contact( "LABELS".scannerOK2 )
      Coil( "DB_INPUTS".inputActive[29] )
   END_RUNG
   // the same network as SCL:
   "DB_INPUTS".activeInputsReqDInt.%X29 := "DB_INPUTS".activeInputsReq[29];
   "DB_INPUTS".inputActive[29] := "LABELS".scannerOK2;
END_REGION

REGION Network 31: A30.- SCANNER UPPER LABLE 2
   RUNG wire#powerrail
      Contact( "DB_INPUTS".activeInputsReq[30] )
      Coil( "DB_INPUTS".activeInputsReqDInt.%X30 )
   END_RUNG
   RUNG wire#powerrail
      Contact( "LABELS".scannerOK4 )
      Coil( "DB_INPUTS".inputActive[30] )
   END_RUNG
   // the same network as SCL:
   "DB_INPUTS".activeInputsReqDInt.%X30 := "DB_INPUTS".activeInputsReq[30];
   "DB_INPUTS".inputActive[30] := "LABELS".scannerOK4;
END_REGION

REGION Network 32: A31.- MANUAL TOOLING ID2
   RUNG wire#powerrail
      Contact( "DB_INPUTS".activeInputsReq[31] )
      Coil( "DB_INPUTS".activeInputsReqDInt.%X31 )
   END_RUNG
   RUNG wire#powerrail
      Contact( "toolingID2" )
      Coil( "DB_INPUTS".inputActive[31] )
   END_RUNG
   // the same network as SCL:
   "DB_INPUTS".activeInputsReqDInt.%X31 := "DB_INPUTS".activeInputsReq[31];
   "DB_INPUTS".inputActive[31] := "toolingID2";
END_REGION

REGION Network 33: HMI SENSOR OVERVIEW
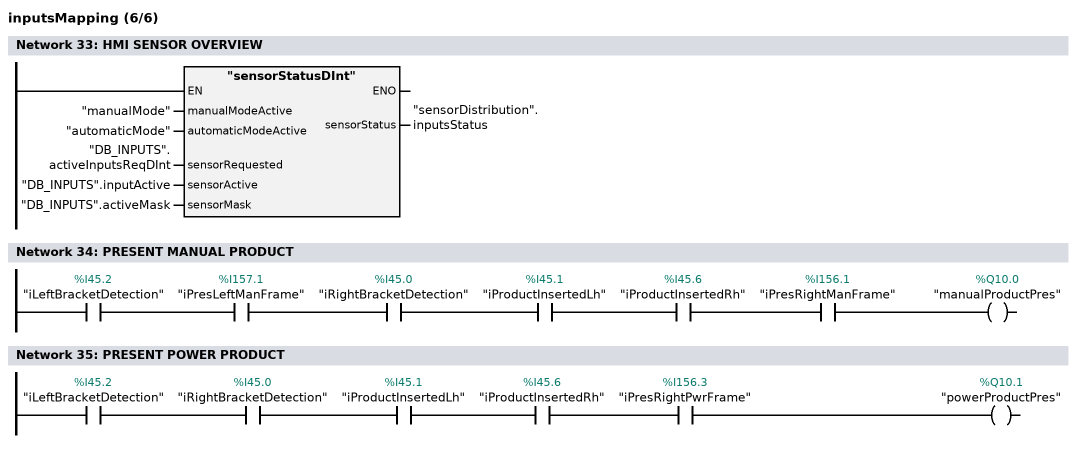
   RUNG wire#powerrail
      "sensorStatusDInt"(manualModeActive := "manualMode", automaticModeActive := "automaticMode", sensorRequested := "DB_INPUTS".activeInputsReqDInt, sensorActive := "DB_INPUTS".inputActive, sensorMask := "DB_INPUTS".activeMask, sensorStatus => "sensorDistribution".inputsStatus)
   END_RUNG
   // the same network as SCL:
   "sensorStatusDInt"(manualModeActive := "manualMode",
                      automaticModeActive := "automaticMode",
                      sensorRequested := "DB_INPUTS".activeInputsReqDInt,
                      sensorActive := "DB_INPUTS".inputActive,
                      sensorMask := "DB_INPUTS".activeMask,
                      sensorStatus => "sensorDistribution".inputsStatus);
END_REGION

REGION Network 34: PRESENT MANUAL PRODUCT
   RUNG wire#powerrail
      Contact( "iLeftBracketDetection" )
      Contact( "iPresLeftManFrame" )
      Contact( "iRightBracketDetection" )
      Contact( "iProductInsertedLh" )
      Contact( "iProductInsertedRh" )
      Contact( "iPresRightManFrame" )
      Coil( "manualProductPres" )
   END_RUNG
   // the same network as SCL:
   "manualProductPres" := "iLeftBracketDetection" AND "iPresLeftManFrame" AND "iRightBracketDetection" AND "iProductInsertedLh" AND "iProductInsertedRh" AND "iPresRightManFrame";
END_REGION

REGION Network 35: PRESENT POWER PRODUCT
   RUNG wire#powerrail
      Contact( "iLeftBracketDetection" )
      Contact( "iRightBracketDetection" )
      Contact( "iProductInsertedLh" )
      Contact( "iProductInsertedRh" )
      Contact( "iPresRightPwrFrame" )
      Coil( "powerProductPres" )
   END_RUNG
   // the same network as SCL:
   "powerProductPres" := "iLeftBracketDetection" AND "iRightBracketDetection" AND "iProductInsertedLh" AND "iProductInsertedRh" AND "iPresRightPwrFrame";
END_REGION
END_FUNCTION

FUNCTION "sensorStatusDInt" : Void   // FC37, LAD
{ S7_Optimized_Access := 'TRUE' }
VERSION : 0.1
// stored: AutoNumber true, IsIECCheckEnabled false, SetENOAutomatically false, UDAEnableTagReadback false
   VAR_INPUT
      manualModeActive : Bool;
      automaticModeActive : Bool;
      sensorRequested : DInt;
      sensorActive : Array[0..31] of Bool;
      sensorMask : Array[0..31] of Bool;
   END_VAR
   VAR_OUTPUT
      sensorStatus : Array[0..31] of Byte;
   END_VAR
BEGIN

REGION Network 1: Status 0
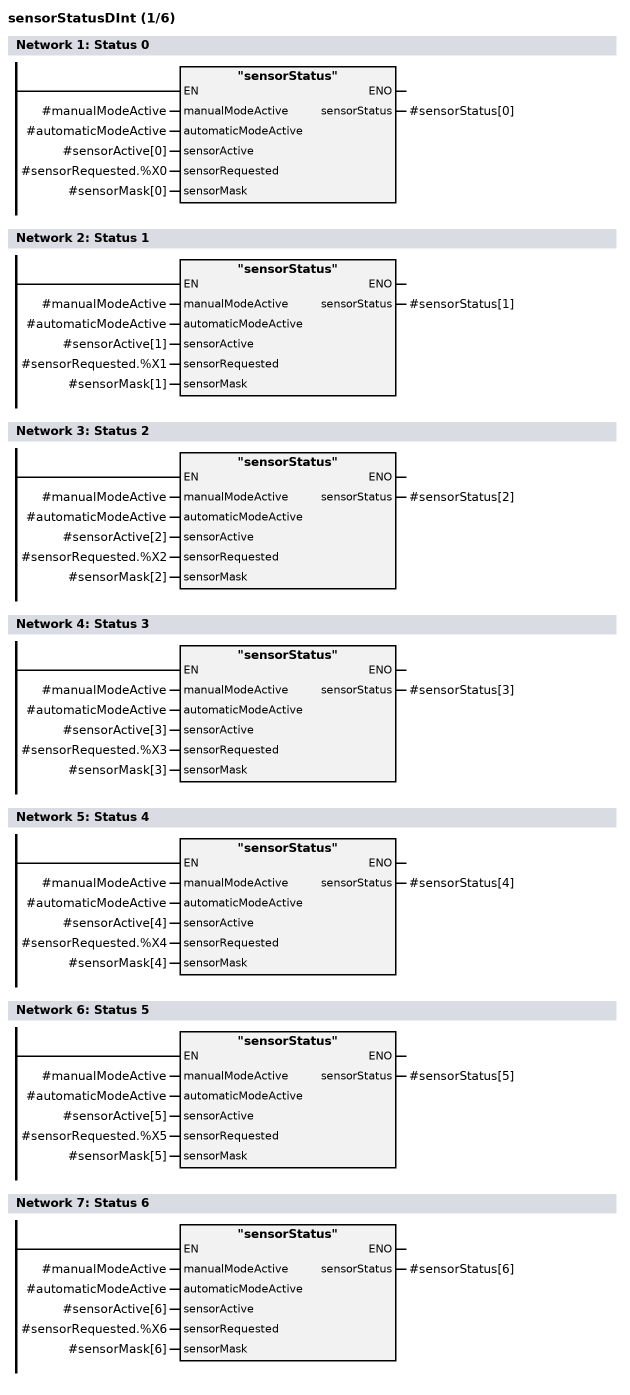
   RUNG wire#powerrail
      "sensorStatus"(manualModeActive := #manualModeActive, automaticModeActive := #automaticModeActive, sensorActive := #sensorActive[0], sensorRequested := #sensorRequested.%X0, sensorMask := #sensorMask[0], sensorStatus => #sensorStatus[0])
   END_RUNG
   // the same network as SCL:
   "sensorStatus"(manualModeActive := #manualModeActive,
                  automaticModeActive := #automaticModeActive,
                  sensorActive := #sensorActive[0],
                  sensorRequested := #sensorRequested.%X0,
                  sensorMask := #sensorMask[0],
                  sensorStatus => #sensorStatus[0]);
END_REGION

REGION Network 2: Status 1
   RUNG wire#powerrail
      "sensorStatus"(manualModeActive := #manualModeActive, automaticModeActive := #automaticModeActive, sensorActive := #sensorActive[1], sensorRequested := #sensorRequested.%X1, sensorMask := #sensorMask[1], sensorStatus => #sensorStatus[1])
   END_RUNG
   // the same network as SCL:
   "sensorStatus"(manualModeActive := #manualModeActive,
                  automaticModeActive := #automaticModeActive,
                  sensorActive := #sensorActive[1],
                  sensorRequested := #sensorRequested.%X1,
                  sensorMask := #sensorMask[1],
                  sensorStatus => #sensorStatus[1]);
END_REGION

REGION Network 3: Status 2
   RUNG wire#powerrail
      "sensorStatus"(manualModeActive := #manualModeActive, automaticModeActive := #automaticModeActive, sensorActive := #sensorActive[2], sensorRequested := #sensorRequested.%X2, sensorMask := #sensorMask[2], sensorStatus => #sensorStatus[2])
   END_RUNG
   // the same network as SCL:
   "sensorStatus"(manualModeActive := #manualModeActive,
                  automaticModeActive := #automaticModeActive,
                  sensorActive := #sensorActive[2],
                  sensorRequested := #sensorRequested.%X2,
                  sensorMask := #sensorMask[2],
                  sensorStatus => #sensorStatus[2]);
END_REGION

REGION Network 4: Status 3
   RUNG wire#powerrail
      "sensorStatus"(manualModeActive := #manualModeActive, automaticModeActive := #automaticModeActive, sensorActive := #sensorActive[3], sensorRequested := #sensorRequested.%X3, sensorMask := #sensorMask[3], sensorStatus => #sensorStatus[3])
   END_RUNG
   // the same network as SCL:
   "sensorStatus"(manualModeActive := #manualModeActive,
                  automaticModeActive := #automaticModeActive,
                  sensorActive := #sensorActive[3],
                  sensorRequested := #sensorRequested.%X3,
                  sensorMask := #sensorMask[3],
                  sensorStatus => #sensorStatus[3]);
END_REGION

REGION Network 5: Status 4
   RUNG wire#powerrail
      "sensorStatus"(manualModeActive := #manualModeActive, automaticModeActive := #automaticModeActive, sensorActive := #sensorActive[4], sensorRequested := #sensorRequested.%X4, sensorMask := #sensorMask[4], sensorStatus => #sensorStatus[4])
   END_RUNG
   // the same network as SCL:
   "sensorStatus"(manualModeActive := #manualModeActive,
                  automaticModeActive := #automaticModeActive,
                  sensorActive := #sensorActive[4],
                  sensorRequested := #sensorRequested.%X4,
                  sensorMask := #sensorMask[4],
                  sensorStatus => #sensorStatus[4]);
END_REGION

REGION Network 6: Status 5
   RUNG wire#powerrail
      "sensorStatus"(manualModeActive := #manualModeActive, automaticModeActive := #automaticModeActive, sensorActive := #sensorActive[5], sensorRequested := #sensorRequested.%X5, sensorMask := #sensorMask[5], sensorStatus => #sensorStatus[5])
   END_RUNG
   // the same network as SCL:
   "sensorStatus"(manualModeActive := #manualModeActive,
                  automaticModeActive := #automaticModeActive,
                  sensorActive := #sensorActive[5],
                  sensorRequested := #sensorRequested.%X5,
                  sensorMask := #sensorMask[5],
                  sensorStatus => #sensorStatus[5]);
END_REGION

REGION Network 7: Status 6
   RUNG wire#powerrail
      "sensorStatus"(manualModeActive := #manualModeActive, automaticModeActive := #automaticModeActive, sensorActive := #sensorActive[6], sensorRequested := #sensorRequested.%X6, sensorMask := #sensorMask[6], sensorStatus => #sensorStatus[6])
   END_RUNG
   // the same network as SCL:
   "sensorStatus"(manualModeActive := #manualModeActive,
                  automaticModeActive := #automaticModeActive,
                  sensorActive := #sensorActive[6],
                  sensorRequested := #sensorRequested.%X6,
                  sensorMask := #sensorMask[6],
                  sensorStatus => #sensorStatus[6]);
END_REGION

REGION Network 8: Status 7
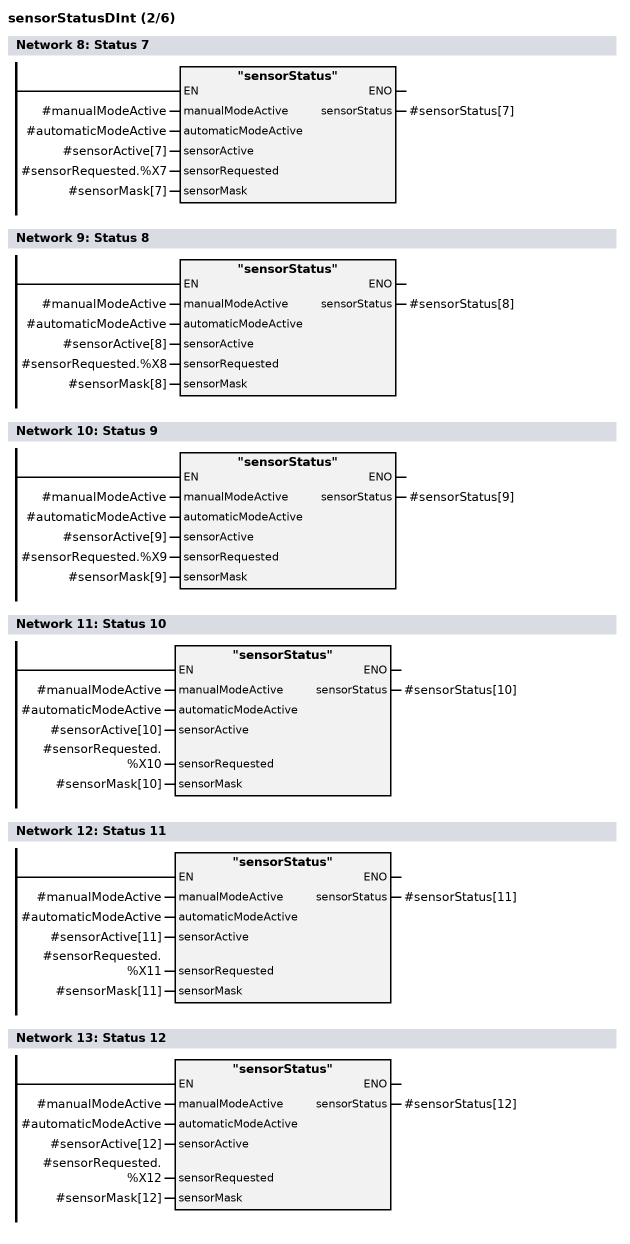
   RUNG wire#powerrail
      "sensorStatus"(manualModeActive := #manualModeActive, automaticModeActive := #automaticModeActive, sensorActive := #sensorActive[7], sensorRequested := #sensorRequested.%X7, sensorMask := #sensorMask[7], sensorStatus => #sensorStatus[7])
   END_RUNG
   // the same network as SCL:
   "sensorStatus"(manualModeActive := #manualModeActive,
                  automaticModeActive := #automaticModeActive,
                  sensorActive := #sensorActive[7],
                  sensorRequested := #sensorRequested.%X7,
                  sensorMask := #sensorMask[7],
                  sensorStatus => #sensorStatus[7]);
END_REGION

REGION Network 9: Status 8
   RUNG wire#powerrail
      "sensorStatus"(manualModeActive := #manualModeActive, automaticModeActive := #automaticModeActive, sensorActive := #sensorActive[8], sensorRequested := #sensorRequested.%X8, sensorMask := #sensorMask[8], sensorStatus => #sensorStatus[8])
   END_RUNG
   // the same network as SCL:
   "sensorStatus"(manualModeActive := #manualModeActive,
                  automaticModeActive := #automaticModeActive,
                  sensorActive := #sensorActive[8],
                  sensorRequested := #sensorRequested.%X8,
                  sensorMask := #sensorMask[8],
                  sensorStatus => #sensorStatus[8]);
END_REGION

REGION Network 10: Status 9
   RUNG wire#powerrail
      "sensorStatus"(manualModeActive := #manualModeActive, automaticModeActive := #automaticModeActive, sensorActive := #sensorActive[9], sensorRequested := #sensorRequested.%X9, sensorMask := #sensorMask[9], sensorStatus => #sensorStatus[9])
   END_RUNG
   // the same network as SCL:
   "sensorStatus"(manualModeActive := #manualModeActive,
                  automaticModeActive := #automaticModeActive,
                  sensorActive := #sensorActive[9],
                  sensorRequested := #sensorRequested.%X9,
                  sensorMask := #sensorMask[9],
                  sensorStatus => #sensorStatus[9]);
END_REGION

REGION Network 11: Status 10
   RUNG wire#powerrail
      "sensorStatus"(manualModeActive := #manualModeActive, automaticModeActive := #automaticModeActive, sensorActive := #sensorActive[10], sensorRequested := #sensorRequested.%X10, sensorMask := #sensorMask[10], sensorStatus => #sensorStatus[10])
   END_RUNG
   // the same network as SCL:
   "sensorStatus"(manualModeActive := #manualModeActive,
                  automaticModeActive := #automaticModeActive,
                  sensorActive := #sensorActive[10],
                  sensorRequested := #sensorRequested.%X10,
                  sensorMask := #sensorMask[10],
                  sensorStatus => #sensorStatus[10]);
END_REGION

REGION Network 12: Status 11
   RUNG wire#powerrail
      "sensorStatus"(manualModeActive := #manualModeActive, automaticModeActive := #automaticModeActive, sensorActive := #sensorActive[11], sensorRequested := #sensorRequested.%X11, sensorMask := #sensorMask[11], sensorStatus => #sensorStatus[11])
   END_RUNG
   // the same network as SCL:
   "sensorStatus"(manualModeActive := #manualModeActive,
                  automaticModeActive := #automaticModeActive,
                  sensorActive := #sensorActive[11],
                  sensorRequested := #sensorRequested.%X11,
                  sensorMask := #sensorMask[11],
                  sensorStatus => #sensorStatus[11]);
END_REGION

REGION Network 13: Status 12
   RUNG wire#powerrail
      "sensorStatus"(manualModeActive := #manualModeActive, automaticModeActive := #automaticModeActive, sensorActive := #sensorActive[12], sensorRequested := #sensorRequested.%X12, sensorMask := #sensorMask[12], sensorStatus => #sensorStatus[12])
   END_RUNG
   // the same network as SCL:
   "sensorStatus"(manualModeActive := #manualModeActive,
                  automaticModeActive := #automaticModeActive,
                  sensorActive := #sensorActive[12],
                  sensorRequested := #sensorRequested.%X12,
                  sensorMask := #sensorMask[12],
                  sensorStatus => #sensorStatus[12]);
END_REGION

REGION Network 14: Status 13
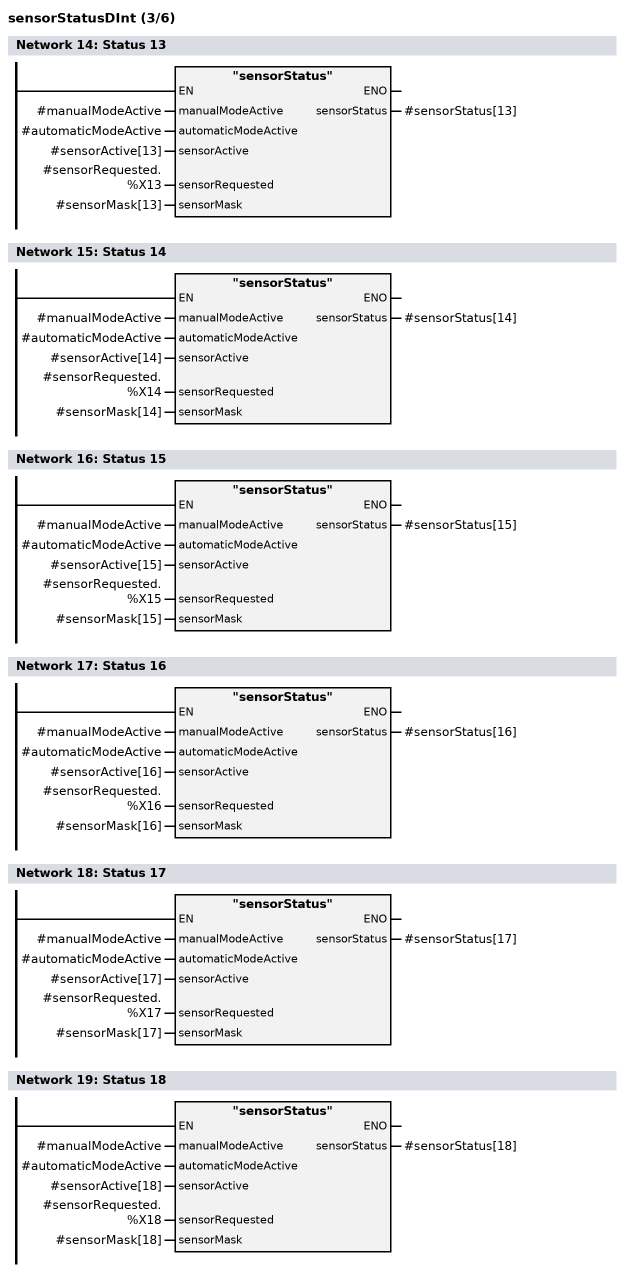
   RUNG wire#powerrail
      "sensorStatus"(manualModeActive := #manualModeActive, automaticModeActive := #automaticModeActive, sensorActive := #sensorActive[13], sensorRequested := #sensorRequested.%X13, sensorMask := #sensorMask[13], sensorStatus => #sensorStatus[13])
   END_RUNG
   // the same network as SCL:
   "sensorStatus"(manualModeActive := #manualModeActive,
                  automaticModeActive := #automaticModeActive,
                  sensorActive := #sensorActive[13],
                  sensorRequested := #sensorRequested.%X13,
                  sensorMask := #sensorMask[13],
                  sensorStatus => #sensorStatus[13]);
END_REGION

REGION Network 15: Status 14
   RUNG wire#powerrail
      "sensorStatus"(manualModeActive := #manualModeActive, automaticModeActive := #automaticModeActive, sensorActive := #sensorActive[14], sensorRequested := #sensorRequested.%X14, sensorMask := #sensorMask[14], sensorStatus => #sensorStatus[14])
   END_RUNG
   // the same network as SCL:
   "sensorStatus"(manualModeActive := #manualModeActive,
                  automaticModeActive := #automaticModeActive,
                  sensorActive := #sensorActive[14],
                  sensorRequested := #sensorRequested.%X14,
                  sensorMask := #sensorMask[14],
                  sensorStatus => #sensorStatus[14]);
END_REGION

REGION Network 16: Status 15
   RUNG wire#powerrail
      "sensorStatus"(manualModeActive := #manualModeActive, automaticModeActive := #automaticModeActive, sensorActive := #sensorActive[15], sensorRequested := #sensorRequested.%X15, sensorMask := #sensorMask[15], sensorStatus => #sensorStatus[15])
   END_RUNG
   // the same network as SCL:
   "sensorStatus"(manualModeActive := #manualModeActive,
                  automaticModeActive := #automaticModeActive,
                  sensorActive := #sensorActive[15],
                  sensorRequested := #sensorRequested.%X15,
                  sensorMask := #sensorMask[15],
                  sensorStatus => #sensorStatus[15]);
END_REGION

REGION Network 17: Status 16
   RUNG wire#powerrail
      "sensorStatus"(manualModeActive := #manualModeActive, automaticModeActive := #automaticModeActive, sensorActive := #sensorActive[16], sensorRequested := #sensorRequested.%X16, sensorMask := #sensorMask[16], sensorStatus => #sensorStatus[16])
   END_RUNG
   // the same network as SCL:
   "sensorStatus"(manualModeActive := #manualModeActive,
                  automaticModeActive := #automaticModeActive,
                  sensorActive := #sensorActive[16],
                  sensorRequested := #sensorRequested.%X16,
                  sensorMask := #sensorMask[16],
                  sensorStatus => #sensorStatus[16]);
END_REGION

REGION Network 18: Status 17
   RUNG wire#powerrail
      "sensorStatus"(manualModeActive := #manualModeActive, automaticModeActive := #automaticModeActive, sensorActive := #sensorActive[17], sensorRequested := #sensorRequested.%X17, sensorMask := #sensorMask[17], sensorStatus => #sensorStatus[17])
   END_RUNG
   // the same network as SCL:
   "sensorStatus"(manualModeActive := #manualModeActive,
                  automaticModeActive := #automaticModeActive,
                  sensorActive := #sensorActive[17],
                  sensorRequested := #sensorRequested.%X17,
                  sensorMask := #sensorMask[17],
                  sensorStatus => #sensorStatus[17]);
END_REGION

REGION Network 19: Status 18
   RUNG wire#powerrail
      "sensorStatus"(manualModeActive := #manualModeActive, automaticModeActive := #automaticModeActive, sensorActive := #sensorActive[18], sensorRequested := #sensorRequested.%X18, sensorMask := #sensorMask[18], sensorStatus => #sensorStatus[18])
   END_RUNG
   // the same network as SCL:
   "sensorStatus"(manualModeActive := #manualModeActive,
                  automaticModeActive := #automaticModeActive,
                  sensorActive := #sensorActive[18],
                  sensorRequested := #sensorRequested.%X18,
                  sensorMask := #sensorMask[18],
                  sensorStatus => #sensorStatus[18]);
END_REGION

REGION Network 20: Status 19
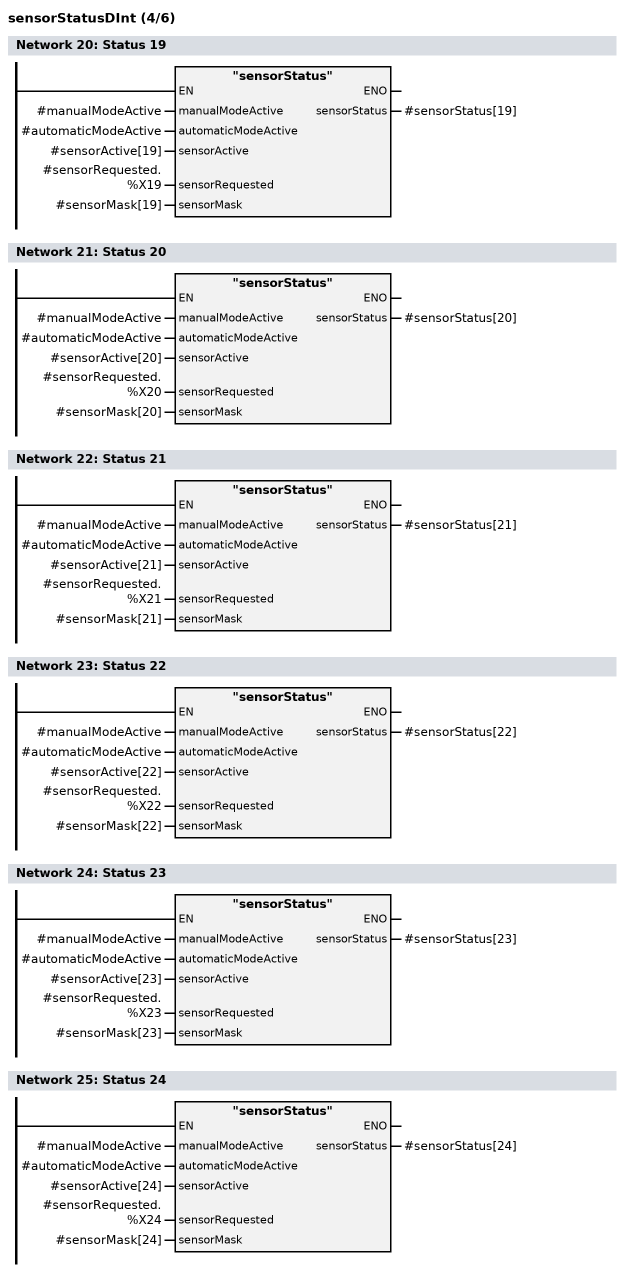
   RUNG wire#powerrail
      "sensorStatus"(manualModeActive := #manualModeActive, automaticModeActive := #automaticModeActive, sensorActive := #sensorActive[19], sensorRequested := #sensorRequested.%X19, sensorMask := #sensorMask[19], sensorStatus => #sensorStatus[19])
   END_RUNG
   // the same network as SCL:
   "sensorStatus"(manualModeActive := #manualModeActive,
                  automaticModeActive := #automaticModeActive,
                  sensorActive := #sensorActive[19],
                  sensorRequested := #sensorRequested.%X19,
                  sensorMask := #sensorMask[19],
                  sensorStatus => #sensorStatus[19]);
END_REGION

REGION Network 21: Status 20
   RUNG wire#powerrail
      "sensorStatus"(manualModeActive := #manualModeActive, automaticModeActive := #automaticModeActive, sensorActive := #sensorActive[20], sensorRequested := #sensorRequested.%X20, sensorMask := #sensorMask[20], sensorStatus => #sensorStatus[20])
   END_RUNG
   // the same network as SCL:
   "sensorStatus"(manualModeActive := #manualModeActive,
                  automaticModeActive := #automaticModeActive,
                  sensorActive := #sensorActive[20],
                  sensorRequested := #sensorRequested.%X20,
                  sensorMask := #sensorMask[20],
                  sensorStatus => #sensorStatus[20]);
END_REGION

REGION Network 22: Status 21
   RUNG wire#powerrail
      "sensorStatus"(manualModeActive := #manualModeActive, automaticModeActive := #automaticModeActive, sensorActive := #sensorActive[21], sensorRequested := #sensorRequested.%X21, sensorMask := #sensorMask[21], sensorStatus => #sensorStatus[21])
   END_RUNG
   // the same network as SCL:
   "sensorStatus"(manualModeActive := #manualModeActive,
                  automaticModeActive := #automaticModeActive,
                  sensorActive := #sensorActive[21],
                  sensorRequested := #sensorRequested.%X21,
                  sensorMask := #sensorMask[21],
                  sensorStatus => #sensorStatus[21]);
END_REGION

REGION Network 23: Status 22
   RUNG wire#powerrail
      "sensorStatus"(manualModeActive := #manualModeActive, automaticModeActive := #automaticModeActive, sensorActive := #sensorActive[22], sensorRequested := #sensorRequested.%X22, sensorMask := #sensorMask[22], sensorStatus => #sensorStatus[22])
   END_RUNG
   // the same network as SCL:
   "sensorStatus"(manualModeActive := #manualModeActive,
                  automaticModeActive := #automaticModeActive,
                  sensorActive := #sensorActive[22],
                  sensorRequested := #sensorRequested.%X22,
                  sensorMask := #sensorMask[22],
                  sensorStatus => #sensorStatus[22]);
END_REGION

REGION Network 24: Status 23
   RUNG wire#powerrail
      "sensorStatus"(manualModeActive := #manualModeActive, automaticModeActive := #automaticModeActive, sensorActive := #sensorActive[23], sensorRequested := #sensorRequested.%X23, sensorMask := #sensorMask[23], sensorStatus => #sensorStatus[23])
   END_RUNG
   // the same network as SCL:
   "sensorStatus"(manualModeActive := #manualModeActive,
                  automaticModeActive := #automaticModeActive,
                  sensorActive := #sensorActive[23],
                  sensorRequested := #sensorRequested.%X23,
                  sensorMask := #sensorMask[23],
                  sensorStatus => #sensorStatus[23]);
END_REGION

REGION Network 25: Status 24
   RUNG wire#powerrail
      "sensorStatus"(manualModeActive := #manualModeActive, automaticModeActive := #automaticModeActive, sensorActive := #sensorActive[24], sensorRequested := #sensorRequested.%X24, sensorMask := #sensorMask[24], sensorStatus => #sensorStatus[24])
   END_RUNG
   // the same network as SCL:
   "sensorStatus"(manualModeActive := #manualModeActive,
                  automaticModeActive := #automaticModeActive,
                  sensorActive := #sensorActive[24],
                  sensorRequested := #sensorRequested.%X24,
                  sensorMask := #sensorMask[24],
                  sensorStatus => #sensorStatus[24]);
END_REGION

REGION Network 26: Status 25
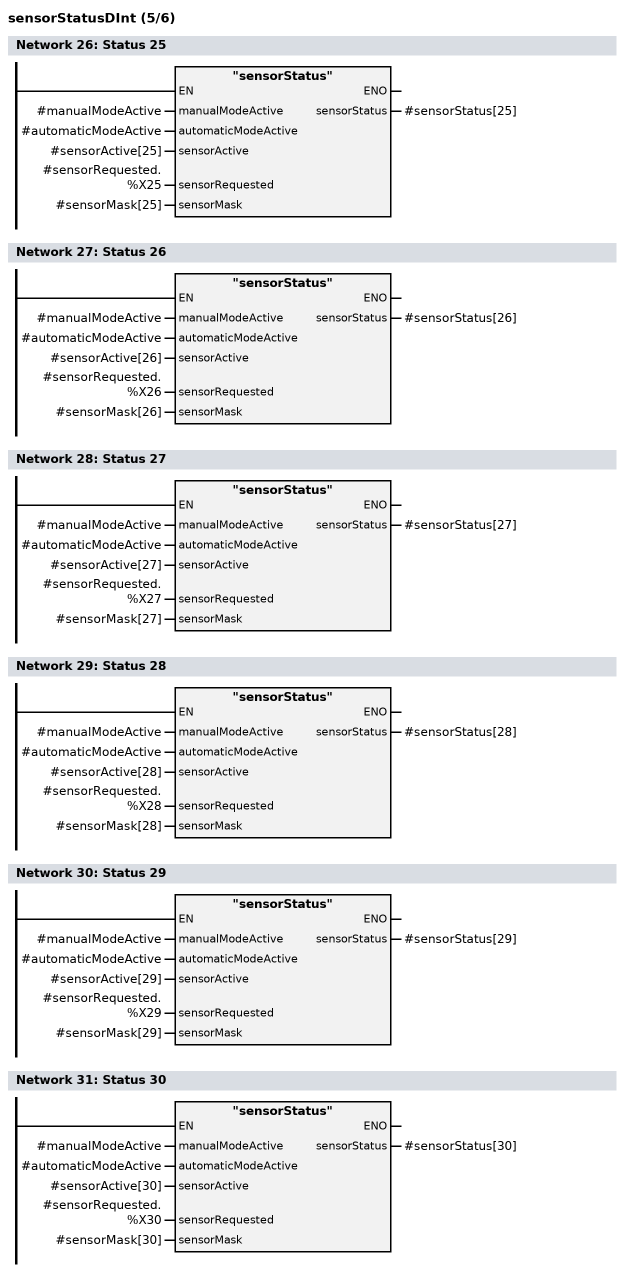
   RUNG wire#powerrail
      "sensorStatus"(manualModeActive := #manualModeActive, automaticModeActive := #automaticModeActive, sensorActive := #sensorActive[25], sensorRequested := #sensorRequested.%X25, sensorMask := #sensorMask[25], sensorStatus => #sensorStatus[25])
   END_RUNG
   // the same network as SCL:
   "sensorStatus"(manualModeActive := #manualModeActive,
                  automaticModeActive := #automaticModeActive,
                  sensorActive := #sensorActive[25],
                  sensorRequested := #sensorRequested.%X25,
                  sensorMask := #sensorMask[25],
                  sensorStatus => #sensorStatus[25]);
END_REGION

REGION Network 27: Status 26
   RUNG wire#powerrail
      "sensorStatus"(manualModeActive := #manualModeActive, automaticModeActive := #automaticModeActive, sensorActive := #sensorActive[26], sensorRequested := #sensorRequested.%X26, sensorMask := #sensorMask[26], sensorStatus => #sensorStatus[26])
   END_RUNG
   // the same network as SCL:
   "sensorStatus"(manualModeActive := #manualModeActive,
                  automaticModeActive := #automaticModeActive,
                  sensorActive := #sensorActive[26],
                  sensorRequested := #sensorRequested.%X26,
                  sensorMask := #sensorMask[26],
                  sensorStatus => #sensorStatus[26]);
END_REGION

REGION Network 28: Status 27
   RUNG wire#powerrail
      "sensorStatus"(manualModeActive := #manualModeActive, automaticModeActive := #automaticModeActive, sensorActive := #sensorActive[27], sensorRequested := #sensorRequested.%X27, sensorMask := #sensorMask[27], sensorStatus => #sensorStatus[27])
   END_RUNG
   // the same network as SCL:
   "sensorStatus"(manualModeActive := #manualModeActive,
                  automaticModeActive := #automaticModeActive,
                  sensorActive := #sensorActive[27],
                  sensorRequested := #sensorRequested.%X27,
                  sensorMask := #sensorMask[27],
                  sensorStatus => #sensorStatus[27]);
END_REGION

REGION Network 29: Status 28
   RUNG wire#powerrail
      "sensorStatus"(manualModeActive := #manualModeActive, automaticModeActive := #automaticModeActive, sensorActive := #sensorActive[28], sensorRequested := #sensorRequested.%X28, sensorMask := #sensorMask[28], sensorStatus => #sensorStatus[28])
   END_RUNG
   // the same network as SCL:
   "sensorStatus"(manualModeActive := #manualModeActive,
                  automaticModeActive := #automaticModeActive,
                  sensorActive := #sensorActive[28],
                  sensorRequested := #sensorRequested.%X28,
                  sensorMask := #sensorMask[28],
                  sensorStatus => #sensorStatus[28]);
END_REGION

REGION Network 30: Status 29
   RUNG wire#powerrail
      "sensorStatus"(manualModeActive := #manualModeActive, automaticModeActive := #automaticModeActive, sensorActive := #sensorActive[29], sensorRequested := #sensorRequested.%X29, sensorMask := #sensorMask[29], sensorStatus => #sensorStatus[29])
   END_RUNG
   // the same network as SCL:
   "sensorStatus"(manualModeActive := #manualModeActive,
                  automaticModeActive := #automaticModeActive,
                  sensorActive := #sensorActive[29],
                  sensorRequested := #sensorRequested.%X29,
                  sensorMask := #sensorMask[29],
                  sensorStatus => #sensorStatus[29]);
END_REGION

REGION Network 31: Status 30
   RUNG wire#powerrail
      "sensorStatus"(manualModeActive := #manualModeActive, automaticModeActive := #automaticModeActive, sensorActive := #sensorActive[30], sensorRequested := #sensorRequested.%X30, sensorMask := #sensorMask[30], sensorStatus => #sensorStatus[30])
   END_RUNG
   // the same network as SCL:
   "sensorStatus"(manualModeActive := #manualModeActive,
                  automaticModeActive := #automaticModeActive,
                  sensorActive := #sensorActive[30],
                  sensorRequested := #sensorRequested.%X30,
                  sensorMask := #sensorMask[30],
                  sensorStatus => #sensorStatus[30]);
END_REGION

REGION Network 32: Status 31
